LIN {X 0,Y 199.613,Z 910.43,A -85,B 0,C 180,E1 -21655.713,E2 -21655.713} C_VEL
LIN {X 0,Y 199.947,Z 910.384,A -85,B 0,C 180,E1 -21661.488,E2 -21661.488} C_VEL
LIN {X 0,Y 200.051,Z 910.436,A -85,B 0,C 180,E1 -21662.505,E2 -21662.505} C_VEL
LIN {X 0,Y 201.275,Z 916.976,A -85,B 0,C 180,E1 -21665.835,E2 -21665.835} C_VEL
LIN {X 0,Y 200.308,Z 922.874,A -85,B 0,C 180,E1 -21668.72,E2 -21668.72} C_VEL
LIN {X 0,Y 200.829,Z 941.062,A -85,B 0,C 180,E1 -21669.859,E2 -21669.859} C_VEL
LIN {X 0,Y 202.996,Z 965.944,A -85,B 0,C 180,E1 -21671.404,E2 -21671.404} C_VEL
LIN {X 0,Y 201.928,Z 1002.393,A -85,B 0,C 180,E1 -21673.768,E2 -21673.768} C_VEL
LIN {X 0,Y 201.253,Z 1013.208,A -85,B 0,C 180,E1 -21674.803,E2 -21674.803} C_VEL
LIN {X 0,Y 200.691,Z 1016.798,A -85,B 0,C 180,E1 -21675.235,E2 -21675.235} C_VEL
LIN {X 0,Y 198.329,Z 1023.524,A -85,B 0,C 180,E1 -21676.228,E2 -21676.228} C_VEL
LIN {X 0,Y 193.611,Z 1034.526,A -85,B 0,C 180,E1 -21678.361,E2 -21678.361} C_VEL
LIN {X 0,Y 192.718,Z 1039.161,A -85,B 0,C 180,E1 -21679.407,E2 -21679.407} C_VEL
LIN {X 0,Y 192.269,Z 1046.284,A -85,B 0,C 180,E1 -21681.169,E2 -21681.169} C_VEL
LIN {X 0,Y 191.944,Z 1053.424,A -85,B 0,C 180,E1 -21683.283,E2 -21683.283} C_VEL
LIN {X 0,Y 191.706,Z 1060.328,A -85,B 0,C 180,E1 -21685.795,E2 -21685.795} C_VEL
LIN {X 0,Y 191.489,Z 1064.888,A -85,B 0,C 180,E1 -21687.896,E2 -21687.896} C_VEL
LIN {X 0,Y 191.203,Z 1070.236,A -85,B 0,C 180,E1 -21691.053,E2 -21691.053} C_VEL
LIN {X 0,Y 190.853,Z 1074.06,A -85,B 0,C 180,E1 -21694.223,E2 -21694.223} C_VEL
LIN {X 0,Y 190.769,Z 1075.958,A -85,B 0,C 180,E1 -21696.345,E2 -21696.345} C_VEL
LIN {X 0,Y 191.01,Z 1077.321,A -85,B 0,C 180,E1 -21698.463,E2 -21698.463} C_VEL
LIN {X 0,Y 191.494,Z 1078.158,A -85,B 0,C 180,E1 -21700.574,E2 -21700.574} C_VEL
LIN {X 0,Y 192.366,Z 1078.612,A -85,B 0,C 180,E1 -21702.662,E2 -21702.662} C_VEL
LIN {X 0,Y 193.533,Z 1078.656,A -85,B 0,C 180,E1 -21704.726,E2 -21704.726} C_VEL
LIN {X 0,Y 195.065,Z 1078.141,A -85,B 0,C 180,E1 -21706.752,E2 -21706.752} C_VEL
LIN {X 0,Y 196.852,Z 1077.188,A -85,B 0,C 180,E1 -21708.742,E2 -21708.742} C_VEL
LIN {X 0,Y 198.954,Z 1075.838,A -85,B 0,C 180,E1 -21710.686,E2 -21710.686} C_VEL
LIN {X 0,Y 202.69,Z 1072.86,A -85,B 0,C 180,E1 -21713.5,E2 -21713.5} C_VEL
LIN {X 0,Y 207.145,Z 1068.693,A -85,B 0,C 180,E1 -21716.171,E2 -21716.171} C_VEL
LIN {X 0,Y 212.234,Z 1063.329,A -85,B 0,C 180,E1 -21718.696,E2 -21718.696} C_VEL
LIN {X 0,Y 217.894,Z 1056.459,A -85,B 0,C 180,E1 -21721.069,E2 -21721.069} C_VEL
LIN {X 0,Y 223.018,Z 1049.383,A -85,B 0,C 180,E1 -21722.929,E2 -21722.929} C_VEL
LIN {X 0,Y 227.532,Z 1042.512,A -85,B 0,C 180,E1 -21724.312,E2 -21724.312} C_VEL
LIN {X 0,Y 232.833,Z 1033.277,A -85,B 0,C 180,E1 -21725.791,E2 -21725.791} C_VEL
LIN {X 0,Y 237.843,Z 1023.421,A -85,B 0,C 180,E1 -21726.993,E2 -21726.993} C_VEL
LIN {X 0,Y 242.457,Z 1012.13,A -85,B 0,C 180,E1 -21728.039,E2 -21728.039} C_VEL
LIN {X 0,Y 246.47,Z 1000.194,A -85,B 0,C 180,E1 -21728.853,E2 -21728.853} C_VEL
LIN {X 0,Y 248.933,Z 990.741,A -85,B 0,C 180,E1 -21729.395,E2 -21729.395} C_VEL
LIN {X 0,Y 248.237,Z 987.091,A -85,B 0,C 180,E1 -21731.284,E2 -21731.284} C_VEL
LIN {X 0,Y 247.848,Z 983.63,A -85,B 0,C 180,E1 -21734.105,E2 -21734.105} C_VEL
LIN {X 0,Y 247.778,Z 983.164,A -85,B 0,C 180,E1 -21735.162,E2 -21735.162} C_VEL
LIN {X 0,Y 248.134,Z 983.137,A -85,B 0,C 180,E1 -21737.635,E2 -21737.635} C_VEL
LIN {X 0,Y 249.346,Z 985.54,A -85,B 0,C 180,E1 -21740.596,E2 -21740.596} C_VEL
LIN {X 0,Y 249.596,Z 986.288,A -85,B 0,C 180,E1 -21741.087,E2 -21741.087} C_VEL
LIN {X 0,Y 246.318,Z 998.437,A -85,B 0,C 180,E1 -21741.85,E2 -21741.85} C_VEL
LIN {X 0,Y 241.936,Z 1011.048,A -85,B 0,C 180,E1 -21742.932,E2 -21742.932} C_VEL
LIN {X 0,Y 237.247,Z 1021.654,A -85,B 0,C 180,E1 -21744.194,E2 -21744.194} C_VEL
LIN {X 0,Y 232.693,Z 1030.307,A -85,B 0,C 180,E1 -21745.508,E2 -21745.508} C_VEL
LIN {X 0,Y 226.976,Z 1039.66,A -85,B 0,C 180,E1 -21747.356,E2 -21747.356} C_VEL
LIN {X 0,Y 222.227,Z 1046.268,A -85,B 0,C 180,E1 -21749.076,E2 -21749.076} C_VEL
LIN {X 0,Y 217.511,Z 1052.076,A -85,B 0,C 180,E1 -21751.01,E2 -21751.01} C_VEL
LIN {X 0,Y 212.195,Z 1057.722,A -85,B 0,C 180,E1 -21753.442,E2 -21753.442} C_VEL
LIN {X 0,Y 207.462,Z 1061.91,A -85,B 0,C 180,E1 -21756.015,E2 -21756.015} C_VEL
LIN {X 0,Y 204.546,Z 1064.015,A -85,B 0,C 180,E1 -21757.794,E2 -21757.794} C_VEL
LIN {X 0,Y 201.845,Z 1065.571,A -85,B 0,C 180,E1 -21759.624,E2 -21759.624} C_VEL
LIN {X 0,Y 199.438,Z 1066.666,A -85,B 0,C 180,E1 -21761.51,E2 -21761.51} C_VEL
LIN {X 0,Y 197.357,Z 1067.342,A -85,B 0,C 180,E1 -21763.449,E2 -21763.449} C_VEL
LIN {X 0,Y 195.619,Z 1067.461,A -85,B 0,C 180,E1 -21765.435,E2 -21765.435} C_VEL
LIN {X 0,Y 194.191,Z 1067.076,A -85,B 0,C 180,E1 -21767.459,E2 -21767.459} C_VEL
LIN {X 0,Y 192.9,Z 1066.286,A -85,B 0,C 180,E1 -21769.505,E2 -21769.505} C_VEL
LIN {X 0,Y 191.826,Z 1065.04,A -85,B 0,C 180,E1 -21771.574,E2 -21771.574} C_VEL
LIN {X 0,Y 190.973,Z 1062.137,A -85,B 0,C 180,E1 -21774.722,E2 -21774.722} C_VEL
LIN {X 0,Y 190.674,Z 1058.072,A -85,B 0,C 180,E1 -21777.889,E2 -21777.889} C_VEL
LIN {X 0,Y 190.619,Z 1052.596,A -85,B 0,C 180,E1 -21781.057,E2 -21781.057} C_VEL
LIN {X 0,Y 190.791,Z 1046.812,A -85,B 0,C 180,E1 -21783.697,E2 -21783.697} C_VEL
LIN {X 0,Y 191.238,Z 1038.6,A -85,B 0,C 180,E1 -21786.649,E2 -21786.649} C_VEL
LIN {X 0,Y 191.776,Z 1030.551,A -85,B 0,C 180,E1 -21788.961,E2 -21788.961} C_VEL
LIN {X 0,Y 192.397,Z 1021.548,A -85,B 0,C 180,E1 -21791.057,E2 -21791.057} C_VEL
LIN {X 0,Y 193.113,Z 1011.82,A -85,B 0,C 180,E1 -21792.881,E2 -21792.881} C_VEL
LIN {X 0,Y 193.848,Z 1001.106,A -85,B 0,C 180,E1 -21794.434,E2 -21794.434} C_VEL
LIN {X 0,Y 194.455,Z 989.47,A -85,B 0,C 180,E1 -21795.729,E2 -21795.729} C_VEL
LIN {X 0,Y 195.048,Z 973.997,A -85,B 0,C 180,E1 -21796.89,E2 -21796.89} C_VEL
LIN {X 0,Y 196.308,Z 933.852,A -85,B 0,C 180,E1 -21799.526,E2 -21799.526} C_VEL
LIN {X 0,Y 193.913,Z 916.288,A -85,B 0,C 180,E1 -21800.666,E2 -21800.666} C_VEL
LIN {X 0,Y 192.915,Z 911.253,A -85,B 0,C 180,E1 -21801.025,E2 -21801.025} C_VEL
LIN {X 0,Y 192.57,Z 911.308,A -85,B 0,C 180,E1 -21805.974,E2 -21805.974} C_VEL
LIN {X 0,Y 192.602,Z 911.303,A -85,B 0,C 180,E1 -21808.866,E2 -21808.866} C_VEL
LIN {X 0,Y 192.596,Z 911.306,A -85,B 0,C 180,E1 -21813.188,E2 -21813.188} C_VEL
LIN {X 0,Y 192.542,Z 911.308,A -85,B 0,C 180,E1 -21818.355,E2 -21818.355} C_VEL
LIN {X 0,Y 192.486,Z 911.319,A -85,B 0,C 180,E1 -21823.094,E2 -21823.094} C_VEL
LIN {X 0,Y 192.488,Z 911.316,A -85,B 0,C 180,E1 -21826.907,E2 -21826.907} C_VEL
LIN {X 0,Y 192.544,Z 911.311,A -85,B 0,C 180,E1 -21831.647,E2 -21831.647} C_VEL
LIN {X 0,Y 192.598,Z 911.301,A -85,B 0,C 180,E1 -21836.814,E2 -21836.814} C_VEL
LIN {X 0,Y 192.624,Z 911.301,A -85,B 0,C 180,E1 -21841.686,E2 -21841.686} C_VEL
LIN {X 0,Y 192.674,Z 911.292,A -85,B 0,C 180,E1 -21846.345,E2 -21846.345} C_VEL
LIN {X 0,Y 192.698,Z 911.294,A -85,B 0,C 180,E1 -21851.492,E2 -21851.492} C_VEL
LIN {X 0,Y 192.74,Z 911.286,A -85,B 0,C 180,E1 -21855.212,E2 -21855.212} C_VEL
LIN {X 0,Y 192.95,Z 911.264,A -85,B 0,C 180,E1 -21859.567,E2 -21859.567} C_VEL
LIN {X 0,Y 192.967,Z 911.258,A -85,B 0,C 180,E1 -21863.728,E2 -21863.728} C_VEL
LIN {X 0,Y 193.212,Z 911.23,A -85,B 0,C 180,E1 -21867.916,E2 -21867.916} C_VEL
LIN {X 0,Y 193.414,Z 911.207,A -85,B 0,C 180,E1 -21870,E2 -21870} C_VEL
LIN {X 0,Y 192.921,Z 911.263,A -85,B 0,C 180,E1 -21874.179,E2 -21874.179} C_VEL
LIN {X 0,Y 193.03,Z 911.254,A -85,B 0,C 180,E1 -21878.374,E2 -21878.374} C_VEL
LIN {X 0,Y 192.781,Z 911.28,A -85,B 0,C 180,E1 -21882.635,E2 -21882.635} C_VEL
LIN {X 0,Y 192.699,Z 911.294,A -85,B 0,C 180,E1 -21888.508,E2 -21888.508} C_VEL
LIN {X 0,Y 192.615,Z 911.299,A -85,B 0,C 180,E1 -21894.189,E2 -21894.189} C_VEL
LIN {X 0,Y 192.605,Z 911.305,A -85,B 0,C 180,E1 -21898.865,E2 -21898.865} C_VEL
LIN {X 0,Y 192.599,Z 911.301,A -85,B 0,C 180,E1 -21903.186,E2 -21903.186} C_VEL
LIN {X 0,Y 192.546,Z 911.311,A -85,B 0,C 180,E1 -21908.354,E2 -21908.354} C_VEL
LIN {X 0,Y 192.49,Z 911.315,A -85,B 0,C 180,E1 -21913.093,E2 -21913.093} C_VEL
LIN {X 0,Y 192.49,Z 911.318,A -85,B 0,C 180,E1 -21916.906,E2 -21916.906} C_VEL
LIN {X 0,Y 192.546,Z 911.307,A -85,B 0,C 180,E1 -21921.645,E2 -21921.645} C_VEL
LIN {X 0,Y 192.598,Z 911.305,A -85,B 0,C 180,E1 -21926.813,E2 -21926.813} C_VEL
LIN {X 0,Y 192.623,Z 911.299,A -85,B 0,C 180,E1 -21931.684,E2 -21931.684} C_VEL
LIN {X 0,Y 192.66,Z 911.297,A -85,B 0,C 180,E1 -21936.341,E2 -21936.341} C_VEL
LIN {X 0,Y 192.698,Z 911.293,A -85,B 0,C 180,E1 -21941.491,E2 -21941.491} C_VEL
LIN {X 0,Y 192.721,Z 911.292,A -85,B 0,C 180,E1 -21945.209,E2 -21945.209} C_VEL
LIN {X 0,Y 192.949,Z 911.26,A -85,B 0,C 180,E1 -21949.566,E2 -21949.566} C_VEL
LIN {X 0,Y 192.965,Z 911.262,A -85,B 0,C 180,E1 -21953.726,E2 -21953.726} C_VEL
LIN {X 0,Y 193.21,Z 911.226,A -85,B 0,C 180,E1 -21957.914,E2 -21957.914} C_VEL
LIN {X 0,Y 193.412,Z 911.204,A -85,B 0,C 180,E1 -21959.999,E2 -21959.999} C_VEL
LIN {X 0,Y 192.918,Z 911.267,A -85,B 0,C 180,E1 -21964.177,E2 -21964.177} C_VEL
LIN {X 0,Y 193.023,Z 911.251,A -85,B 0,C 180,E1 -21968.373,E2 -21968.373} C_VEL
LIN {X 0,Y 192.782,Z 911.284,A -85,B 0,C 180,E1 -21972.634,E2 -21972.634} C_VEL
LIN {X 0,Y 192.704,Z 911.291,A -85,B 0,C 180,E1 -21976.963,E2 -21976.963} C_VEL
LIN {X 0,Y 192.573,Z 911.309,A -85,B 0,C 180,E1 -21981.404,E2 -21981.404} C_VEL
LIN {X 0,Y 192.611,Z 911.3,A -85,B 0,C 180,E1 -21984.188,E2 -21984.188} C_VEL
LIN {X 0,Y 192.601,Z 911.305,A -85,B 0,C 180,E1 -21988.864,E2 -21988.864} C_VEL
LIN {X 0,Y 192.595,Z 911.306,A -85,B 0,C 180,E1 -21993.186,E2 -21993.186} C_VEL
LIN {X 0,Y 192.541,Z 911.312,A -85,B 0,C 180,E1 -21998.353,E2 -21998.353} C_VEL
LIN {X 0,Y 192.485,Z 911.315,A -85,B 0,C 180,E1 -22003.093,E2 -22003.093} C_VEL
LIN {X 0,Y 192.485,Z 911.318,A -85,B 0,C 180,E1 -22006.905,E2 -22006.905} C_VEL
LIN {X 0,Y 192.541,Z 911.31,A -85,B 0,C 180,E1 -22011.645,E2 -22011.645} C_VEL
LIN {X 0,Y 192.599,Z 911.307,A -85,B 0,C 180,E1 -22016.814,E2 -22016.814} C_VEL
LIN {X 0,Y 193.061,Z 911.351,A -85,B 0,C 180,E1 -22022.786,E2 -22022.786} C_VEL
LIN {X 0,Y 194.169,Z 916.994,A -85,B 0,C 180,E1 -22025.773,E2 -22025.773} C_VEL
LIN {X 0,Y 193.24,Z 922.433,A -85,B 0,C 180,E1 -22028.602,E2 -22028.602} C_VEL
LIN {X 0,Y 193.68,Z 940.397,A -85,B 0,C 180,E1 -22029.776,E2 -22029.776} C_VEL
LIN {X 0,Y 195.896,Z 965.867,A -85,B 0,C 180,E1 -22031.433,E2 -22031.433} C_VEL
LIN {X 0,Y 194.873,Z 1001.979,A -85,B 0,C 180,E1 -22033.904,E2 -22033.904} C_VEL
LIN {X 0,Y 194.128,Z 1014.314,A -85,B 0,C 180,E1 -22035.185,E2 -22035.185} C_VEL
LIN {X 0,Y 193.646,Z 1024.555,A -85,B 0,C 180,E1 -22036.622,E2 -22036.622} C_VEL
LIN {X 0,Y 192.992,Z 1034.779,A -85,B 0,C 180,E1 -22038.446,E2 -22038.446} C_VEL
LIN {X 0,Y 192.718,Z 1039.161,A -85,B 0,C 180,E1 -22039.407,E2 -22039.407} C_VEL
LIN {X 0,Y 191.84,Z 1043.702,A -85,B 0,C 180,E1 -22040.518,E2 -22040.518} C_VEL
LIN {X 0,Y 190.093,Z 1047.709,A -85,B 0,C 180,E1 -22041.719,E2 -22041.719} C_VEL
LIN {X 0,Y 185.624,Z 1056.056,A -85,B 0,C 180,E1 -22044.869,E2 -22044.869} C_VEL
LIN {X 0,Y 184.797,Z 1059.5,A -85,B 0,C 180,E1 -22046.348,E2 -22046.348} C_VEL
LIN {X 0,Y 184.526,Z 1064.875,A -85,B 0,C 180,E1 -22048.908,E2 -22048.908} C_VEL
LIN {X 0,Y 184.314,Z 1068.52,A -85,B 0,C 180,E1 -22051.092,E2 -22051.092} C_VEL
LIN {X 0,Y 183.898,Z 1072.684,A -85,B 0,C 180,E1 -22054.383,E2 -22054.383} C_VEL
LIN {X 0,Y 183.818,Z 1074.699,A -85,B 0,C 180,E1 -22056.586,E2 -22056.586} C_VEL
LIN {X 0,Y 184.05,Z 1076.245,A -85,B 0,C 180,E1 -22058.785,E2 -22058.785} C_VEL
LIN {X 0,Y 184.551,Z 1077.372,A -85,B 0,C 180,E1 -22060.976,E2 -22060.976} C_VEL
LIN {X 0,Y 185.461,Z 1078.068,A -85,B 0,C 180,E1 -22063.142,E2 -22063.142} C_VEL
LIN {X 0,Y 186.677,Z 1078.217,A -85,B 0,C 180,E1 -22065.28,E2 -22065.28} C_VEL
LIN {X 0,Y 190.141,Z 1077.365,A -85,B 0,C 180,E1 -22069.43,E2 -22069.43} C_VEL
LIN {X 0,Y 192.337,Z 1076.209,A -85,B 0,C 180,E1 -22071.432,E2 -22071.432} C_VEL
LIN {X 0,Y 196.255,Z 1073.673,A -85,B 0,C 180,E1 -22074.319,E2 -22074.319} C_VEL
LIN {X 0,Y 200.896,Z 1070.053,A -85,B 0,C 180,E1 -22077.051,E2 -22077.051} C_VEL
LIN {X 0,Y 206.16,Z 1065.117,A -85,B 0,C 180,E1 -22079.624,E2 -22079.624} C_VEL
LIN {X 0,Y 210.987,Z 1060.06,A -85,B 0,C 180,E1 -22081.643,E2 -22081.643} C_VEL
LIN {X 0,Y 216.211,Z 1053.859,A -85,B 0,C 180,E1 -22083.545,E2 -22083.545} C_VEL
LIN {X 0,Y 221.935,Z 1046.324,A -85,B 0,C 180,E1 -22085.304,E2 -22085.304} C_VEL
LIN {X 0,Y 228.294,Z 1036.758,A -85,B 0,C 180,E1 -22087.002,E2 -22087.002} C_VEL
LIN {X 0,Y 233.954,Z 1026.535,A -85,B 0,C 180,E1 -22088.323,E2 -22088.323} C_VEL
LIN {X 0,Y 239.092,Z 1015.776,A -85,B 0,C 180,E1 -22089.395,E2 -22089.395} C_VEL
LIN {X 0,Y 243.435,Z 1004.387,A -85,B 0,C 180,E1 -22090.233,E2 -22090.233} C_VEL
LIN {X 0,Y 246.188,Z 995.227,A -85,B 0,C 180,E1 -22090.794,E2 -22090.794} C_VEL
LIN {X 0,Y 246.017,Z 993.347,A -85,B 0,C 180,E1 -22091.921,E2 -22091.921} C_VEL
LIN {X 0,Y 245.926,Z 990.354,A -85,B 0,C 180,E1 -22094.403,E2 -22094.403} C_VEL
LIN {X 0,Y 246.067,Z 989.856,A -85,B 0,C 180,E1 -22096.728,E2 -22096.728} C_VEL
LIN {X 0,Y 246.307,Z 990.295,A -85,B 0,C 180,E1 -22098.048,E2 -22098.048} C_VEL
LIN {X 0,Y 246.851,Z 991.576,A -85,B 0,C 180,E1 -22099.769,E2 -22099.769} C_VEL
LIN {X 0,Y 242.902,Z 1004.222,A -85,B 0,C 180,E1 -22100.622,E2 -22100.622} C_VEL
LIN {X 0,Y 238.748,Z 1014.42,A -85,B 0,C 180,E1 -22101.588,E2 -22101.588} C_VEL
LIN {X 0,Y 233.909,Z 1024.259,A -85,B 0,C 180,E1 -22102.796,E2 -22102.796} C_VEL
LIN {X 0,Y 228.57,Z 1033.478,A -85,B 0,C 180,E1 -22104.254,E2 -22104.254} C_VEL
LIN {X 0,Y 224.029,Z 1040.184,A -85,B 0,C 180,E1 -22105.621,E2 -22105.621} C_VEL
LIN {X 0,Y 218.648,Z 1047.117,A -85,B 0,C 180,E1 -22107.426,E2 -22107.426} C_VEL
LIN {X 0,Y 213.847,Z 1052.566,A -85,B 0,C 180,E1 -22109.218,E2 -22109.218} C_VEL
LIN {X 0,Y 207.879,Z 1058.36,A -85,B 0,C 180,E1 -22111.751,E2 -22111.751} C_VEL
LIN {X 0,Y 202.523,Z 1062.642,A -85,B 0,C 180,E1 -22114.456,E2 -22114.456} C_VEL
LIN {X 0,Y 198.095,Z 1065.348,A -85,B 0,C 180,E1 -22117.03,E2 -22117.03} C_VEL
LIN {X 0,Y 195.309,Z 1066.722,A -85,B 0,C 180,E1 -22118.911,E2 -22118.911} C_VEL
LIN {X 0,Y 192.768,Z 1067.514,A -85,B 0,C 180,E1 -22120.846,E2 -22120.846} C_VEL
LIN {X 0,Y 190.602,Z 1067.84,A -85,B 0,C 180,E1 -22122.845,E2 -22122.845} C_VEL
LIN {X 0,Y 188.778,Z 1067.767,A -85,B 0,C 180,E1 -22124.895,E2 -22124.895} C_VEL
LIN {X 0,Y 187.286,Z 1067.222,A -85,B 0,C 180,E1 -22126.989,E2 -22126.989} C_VEL
LIN {X 0,Y 185.935,Z 1066.121,A -85,B 0,C 180,E1 -22129.107,E2 -22129.107} C_VEL
LIN {X 0,Y 184.643,Z 1064.185,A -85,B 0,C 180,E1 -22131.74,E2 -22131.74} C_VEL
LIN {X 0,Y 183.951,Z 1061.382,A -85,B 0,C 180,E1 -22134.52,E2 -22134.52} C_VEL
LIN {X 0,Y 183.674,Z 1056.99,A -85,B 0,C 180,E1 -22137.808,E2 -22137.808} C_VEL
LIN {X 0,Y 183.649,Z 1051.201,A -85,B 0,C 180,E1 -22141.097,E2 -22141.097} C_VEL
LIN {X 0,Y 183.837,Z 1044.932,A -85,B 0,C 180,E1 -22143.837,E2 -22143.837} C_VEL
LIN {X 0,Y 184.283,Z 1037.182,A -85,B 0,C 180,E1 -22146.571,E2 -22146.571} C_VEL
LIN {X 0,Y 184.847,Z 1028.643,A -85,B 0,C 180,E1 -22149.024,E2 -22149.024} C_VEL
LIN {X 0,Y 185.591,Z 1017.821,A -85,B 0,C 180,E1 -22151.468,E2 -22151.468} C_VEL
LIN {X 0,Y 186.206,Z 1008.819,A -85,B 0,C 180,E1 -22153.09,E2 -22153.09} C_VEL
LIN {X 0,Y 186.966,Z 997.471,A -85,B 0,C 180,E1 -22154.699,E2 -22154.699} C_VEL
LIN {X 0,Y 187.473,Z 985.392,A -85,B 0,C 180,E1 -22155.911,E2 -22155.911} C_VEL
LIN {X 0,Y 188.831,Z 947.508,A -85,B 0,C 180,E1 -22158.584,E2 -22158.584} C_VEL
LIN {X 0,Y 189.199,Z 934.016,A -85,B 0,C 180,E1 -22159.506,E2 -22159.506} C_VEL
LIN {X 0,Y 186.804,Z 916.793,A -85,B 0,C 180,E1 -22160.665,E2 -22160.665} C_VEL
LIN {X 0,Y 185.884,Z 912.129,A -85,B 0,C 180,E1 -22161.027,E2 -22161.027} C_VEL
LIN {X 0,Y 185.509,Z 912.19,A -85,B 0,C 180,E1 -22167.042,E2 -22167.042} C_VEL
LIN {X 0,Y 185.545,Z 912.18,A -85,B 0,C 180,E1 -22169.5,E2 -22169.5} C_VEL
LIN {X 0,Y 185.498,Z 912.189,A -85,B 0,C 180,E1 -22174.634,E2 -22174.634} C_VEL
LIN {X 0,Y 185.501,Z 912.189,A -85,B 0,C 180,E1 -22177.316,E2 -22177.316} C_VEL
LIN {X 0,Y 185.462,Z 912.191,A -85,B 0,C 180,E1 -22180.722,E2 -22180.722} C_VEL
LIN {X 0,Y 185.458,Z 912.195,A -85,B 0,C 180,E1 -22186.057,E2 -22186.057} C_VEL
LIN {X 0,Y 185.459,Z 912.192,A -85,B 0,C 180,E1 -22189.893,E2 -22189.893} C_VEL
LIN {X 0,Y 185.503,Z 912.19,A -85,B 0,C 180,E1 -22192.715,E2 -22192.715} C_VEL
LIN {X 0,Y 185.534,Z 912.18,A -85,B 0,C 180,E1 -22197.973,E2 -22197.973} C_VEL
LIN {X 0,Y 185.55,Z 912.184,A -85,B 0,C 180,E1 -22200.596,E2 -22200.596} C_VEL
LIN {X 0,Y 185.584,Z 912.176,A -85,B 0,C 180,E1 -22205.382,E2 -22205.382} C_VEL
LIN {X 0,Y 185.629,Z 912.176,A -85,B 0,C 180,E1 -22211.179,E2 -22211.179} C_VEL
LIN {X 0,Y 185.669,Z 912.166,A -85,B 0,C 180,E1 -22214.635,E2 -22214.635} C_VEL
LIN {X 0,Y 185.893,Z 912.142,A -85,B 0,C 180,E1 -22219.419,E2 -22219.419} C_VEL
LIN {X 0,Y 185.933,Z 912.136,A -85,B 0,C 180,E1 -22223.489,E2 -22223.489} C_VEL
LIN {X 0,Y 186.379,Z 912.083,A -85,B 0,C 180,E1 -22230,E2 -22230} C_VEL
LIN {X 0,Y 185.932,Z 912.136,A -85,B 0,C 180,E1 -22236.512,E2 -22236.512} C_VEL
LIN {X 0,Y 185.893,Z 912.142,A -85,B 0,C 180,E1 -22240.581,E2 -22240.581} C_VEL
LIN {X 0,Y 185.646,Z 912.169,A -85,B 0,C 180,E1 -22245.367,E2 -22245.367} C_VEL
LIN {X 0,Y 185.629,Z 912.176,A -85,B 0,C 180,E1 -22248.821,E2 -22248.821} C_VEL
LIN {X 0,Y 185.549,Z 912.18,A -85,B 0,C 180,E1 -22254.624,E2 -22254.624} C_VEL
LIN {X 0,Y 185.548,Z 912.184,A -85,B 0,C 180,E1 -22259.499,E2 -22259.499} C_VEL
LIN {X 0,Y 185.501,Z 912.187,A -85,B 0,C 180,E1 -22264.632,E2 -22264.632} C_VEL
LIN {X 0,Y 185.504,Z 912.19,A -85,B 0,C 180,E1 -22267.314,E2 -22267.314} C_VEL
LIN {X 0,Y 185.466,Z 912.189,A -85,B 0,C 180,E1 -22270.721,E2 -22270.721} C_VEL
LIN {X 0,Y 185.46,Z 912.197,A -85,B 0,C 180,E1 -22276.055,E2 -22276.055} C_VEL
LIN {X 0,Y 185.461,Z 912.193,A -85,B 0,C 180,E1 -22279.892,E2 -22279.892} C_VEL
LIN {X 0,Y 185.504,Z 912.189,A -85,B 0,C 180,E1 -22282.713,E2 -22282.713} C_VEL
LIN {X 0,Y 185.534,Z 912.184,A -85,B 0,C 180,E1 -22287.972,E2 -22287.972} C_VEL
LIN {X 0,Y 185.55,Z 912.18,A -85,B 0,C 180,E1 -22290.595,E2 -22290.595} C_VEL
LIN {X 0,Y 185.548,Z 912.184,A -85,B 0,C 180,E1 -22295.376,E2 -22295.376} C_VEL
LIN {X 0,Y 185.628,Z 912.173,A -85,B 0,C 180,E1 -22301.178,E2 -22301.178} C_VEL
LIN {X 0,Y 185.707,Z 912.162,A -85,B 0,C 180,E1 -22306.874,E2 -22306.874} C_VEL
LIN {X 0,Y 185.978,Z 912.13,A -85,B 0,C 180,E1 -22311.305,E2 -22311.305} C_VEL
LIN {X 0,Y 186.158,Z 912.104,A -85,B 0,C 180,E1 -22317.835,E2 -22317.835} C_VEL
LIN {X 0,Y 186.377,Z 912.08,A -85,B 0,C 180,E1 -22319.999,E2 -22319.999} C_VEL
LIN {X 0,Y 185.927,Z 912.133,A -85,B 0,C 180,E1 -22326.51,E2 -22326.51} C_VEL
LIN {X 0,Y 185.89,Z 912.143,A -85,B 0,C 180,E1 -22330.58,E2 -22330.58} C_VEL
LIN {X 0,Y 185.652,Z 912.166,A -85,B 0,C 180,E1 -22335.365,E2 -22335.365} C_VEL
LIN {X 0,Y 185.626,Z 912.174,A -85,B 0,C 180,E1 -22338.82,E2 -22338.82} C_VEL
LIN {X 0,Y 185.545,Z 912.181,A -85,B 0,C 180,E1 -22344.622,E2 -22344.622} C_VEL
LIN {X 0,Y 185.544,Z 912.186,A -85,B 0,C 180,E1 -22349.498,E2 -22349.498} C_VEL
LIN {X 0,Y 185.497,Z 912.184,A -85,B 0,C 180,E1 -22354.631,E2 -22354.631} C_VEL
LIN {X 0,Y 185.499,Z 912.189,A -85,B 0,C 180,E1 -22357.314,E2 -22357.314} C_VEL
LIN {X 0,Y 185.462,Z 912.193,A -85,B 0,C 180,E1 -22360.72,E2 -22360.72} C_VEL
LIN {X 0,Y 185.456,Z 912.195,A -85,B 0,C 180,E1 -22366.055,E2 -22366.055} C_VEL
LIN {X 0,Y 185.456,Z 912.196,A -85,B 0,C 180,E1 -22369.891,E2 -22369.891} C_VEL
LIN {X 0,Y 185.499,Z 912.185,A -85,B 0,C 180,E1 -22372.713,E2 -22372.713} C_VEL
LIN {X 0,Y 185.575,Z 912.18,A -85,B 0,C 180,E1 -22377.98,E2 -22377.98} C_VEL
LIN {X 0,Y 186.041,Z 912.134,A -85,B 0,C 180,E1 -22383.043,E2 -22383.043} C_VEL
LIN {X 0,Y 186.989,Z 916.741,A -85,B 0,C 180,E1 -22385.579,E2 -22385.579} C_VEL
LIN {X 0,Y 186.152,Z 922.334,A -85,B 0,C 180,E1 -22388.547,E2 -22388.547} C_VEL
LIN {X 0,Y 186.629,Z 941.521,A -85,B 0,C 180,E1 -22389.867,E2 -22389.867} C_VEL
LIN {X 0,Y 188.81,Z 966.35,A -85,B 0,C 180,E1 -22391.555,E2 -22391.555} C_VEL
LIN {X 0,Y 187.807,Z 1001.86,A -85,B 0,C 180,E1 -22394.118,E2 -22394.118} C_VEL
LIN {X 0,Y 187.082,Z 1014.101,A -85,B 0,C 180,E1 -22395.45,E2 -22395.45} C_VEL
LIN {X 0,Y 186.609,Z 1024.295,A -85,B 0,C 180,E1 -22396.94,E2 -22396.94} C_VEL
LIN {X 0,Y 185.971,Z 1034.491,A -85,B 0,C 180,E1 -22398.832,E2 -22398.832} C_VEL
LIN {X 0,Y 185.473,Z 1042.984,A -85,B 0,C 180,E1 -22400.843,E2 -22400.843} C_VEL
LIN {X 0,Y 185.117,Z 1050.175,A -85,B 0,C 180,E1 -22402.935,E2 -22402.935} C_VEL
LIN {X 0,Y 184.915,Z 1056.366,A -85,B 0,C 180,E1 -22405.094,E2 -22405.094} C_VEL
LIN {X 0,Y 184.797,Z 1059.5,A -85,B 0,C 180,E1 -22406.348,E2 -22406.348} C_VEL
LIN {X 0,Y 183.946,Z 1062.661,A -85,B 0,C 180,E1 -22407.871,E2 -22407.871} C_VEL
LIN {X 0,Y 182.207,Z 1065.218,A -85,B 0,C 180,E1 -22409.462,E2 -22409.462} C_VEL
LIN {X 0,Y 178.237,Z 1069.314,A -85,B 0,C 180,E1 -22412.853,E2 -22412.853} C_VEL
LIN {X 0,Y 177.065,Z 1071.181,A -85,B 0,C 180,E1 -22414.66,E2 -22414.66} C_VEL
LIN {X 0,Y 176.93,Z 1071.85,A -85,B 0,C 180,E1 -22415.27,E2 -22415.27} C_VEL
LIN {X 0,Y 177.131,Z 1075.134,A -85,B 0,C 180,E1 -22419.131,E2 -22419.131} C_VEL
LIN {X 0,Y 177.645,Z 1076.441,A -85,B 0,C 180,E1 -22421.409,E2 -22421.409} C_VEL
LIN {X 0,Y 179.844,Z 1077.726,A -85,B 0,C 180,E1 -22425.875,E2 -22425.875} C_VEL
LIN {X 0,Y 181.515,Z 1077.786,A -85,B 0,C 180,E1 -22428.044,E2 -22428.044} C_VEL
LIN {X 0,Y 185.748,Z 1076.415,A -85,B 0,C 180,E1 -22432.232,E2 -22432.232} C_VEL
LIN {X 0,Y 188.366,Z 1075.181,A -85,B 0,C 180,E1 -22434.231,E2 -22434.231} C_VEL
LIN {X 0,Y 193.011,Z 1072.32,A -85,B 0,C 180,E1 -22437.075,E2 -22437.075} C_VEL
LIN {X 0,Y 198.268,Z 1068.366,A -85,B 0,C 180,E1 -22439.752,E2 -22439.752} C_VEL
LIN {X 0,Y 204.114,Z 1063.197,A -85,B 0,C 180,E1 -22442.255,E2 -22442.255} C_VEL
LIN {X 0,Y 211.688,Z 1055.492,A -85,B 0,C 180,E1 -22444.938,E2 -22444.938} C_VEL
LIN {X 0,Y 217.638,Z 1048.375,A -85,B 0,C 180,E1 -22446.684,E2 -22446.684} C_VEL
LIN {X 0,Y 224.464,Z 1039.022,A -85,B 0,C 180,E1 -22448.428,E2 -22448.428} C_VEL
LIN {X 0,Y 230.685,Z 1029.152,A -85,B 0,C 180,E1 -22449.775,E2 -22449.775} C_VEL
LIN {X 0,Y 236.796,Z 1017.209,A -85,B 0,C 180,E1 -22450.974,E2 -22450.974} C_VEL
LIN {X 0,Y 241.585,Z 1006.027,A -85,B 0,C 180,E1 -22451.811,E2 -22451.811} C_VEL
LIN {X 0,Y 243.512,Z 1000.473,A -85,B 0,C 180,E1 -22452.13,E2 -22452.13} C_VEL
LIN {X 0,Y 243.617,Z 999.565,A -85,B 0,C 180,E1 -22452.534,E2 -22452.534} C_VEL
LIN {X 0,Y 243.682,Z 997.94,A -85,B 0,C 180,E1 -22453.862,E2 -22453.862} C_VEL
LIN {X 0,Y 243.888,Z 996.666,A -85,B 0,C 180,E1 -22456.244,E2 -22456.244} C_VEL
LIN {X 0,Y 244.204,Z 997.405,A -85,B 0,C 180,E1 -22458.44,E2 -22458.44} C_VEL
LIN {X 0,Y 240.203,Z 1008.138,A -85,B 0,C 180,E1 -22459.233,E2 -22459.233} C_VEL
LIN {X 0,Y 235.252,Z 1018.903,A -85,B 0,C 180,E1 -22460.316,E2 -22460.316} C_VEL
LIN {X 0,Y 229.487,Z 1029.124,A -85,B 0,C 180,E1 -22461.674,E2 -22461.674} C_VEL
LIN {X 0,Y 224.556,Z 1036.55,A -85,B 0,C 180,E1 -22462.954,E2 -22462.954} C_VEL
LIN {X 0,Y 217.528,Z 1045.679,A -85,B 0,C 180,E1 -22465.008,E2 -22465.008} C_VEL
LIN {X 0,Y 211.983,Z 1051.678,A -85,B 0,C 180,E1 -22466.837,E2 -22466.837} C_VEL
LIN {X 0,Y 205.792,Z 1057.434,A -85,B 0,C 180,E1 -22469.186,E2 -22469.186} C_VEL
LIN {X 0,Y 200.896,Z 1061.269,A -85,B 0,C 180,E1 -22471.28,E2 -22471.28} C_VEL
LIN {X 0,Y 194.89,Z 1065.127,A -85,B 0,C 180,E1 -22474.36,E2 -22474.36} C_VEL
LIN {X 0,Y 191.695,Z 1066.597,A -85,B 0,C 180,E1 -22476.217,E2 -22476.217} C_VEL
LIN {X 0,Y 188.77,Z 1067.618,A -85,B 0,C 180,E1 -22478.143,E2 -22478.143} C_VEL
LIN {X 0,Y 186.131,Z 1068.231,A -85,B 0,C 180,E1 -22480.135,E2 -22480.135} C_VEL
LIN {X 0,Y 183.855,Z 1068.337,A -85,B 0,C 180,E1 -22482.194,E2 -22482.194} C_VEL
LIN {X 0,Y 180.383,Z 1067.112,A -85,B 0,C 180,E1 -22486.482,E2 -22486.482} C_VEL
LIN {X 0,Y 178.987,Z 1065.887,A -85,B 0,C 180,E1 -22488.679,E2 -22488.679} C_VEL
LIN {X 0,Y 177.524,Z 1063.295,A -85,B 0,C 180,E1 -22491.778,E2 -22491.778} C_VEL
LIN {X 0,Y 176.794,Z 1059.06,A -85,B 0,C 180,E1 -22495.441,E2 -22495.441} C_VEL
LIN {X 0,Y 176.625,Z 1053.778,A -85,B 0,C 180,E1 -22498.861,E2 -22498.861} C_VEL
LIN {X 0,Y 176.785,Z 1047.015,A -85,B 0,C 180,E1 -22502.279,E2 -22502.279} C_VEL
LIN {X 0,Y 177.117,Z 1038.771,A -85,B 0,C 180,E1 -22505.467,E2 -22505.467} C_VEL
LIN {X 0,Y 177.6,Z 1031.527,A -85,B 0,C 180,E1 -22507.735,E2 -22507.735} C_VEL
LIN {X 0,Y 178.262,Z 1021.803,A -85,B 0,C 180,E1 -22510.22,E2 -22510.22} C_VEL
LIN {X 0,Y 179.067,Z 1010.463,A -85,B 0,C 180,E1 -22512.467,E2 -22512.467} C_VEL
LIN {X 0,Y 179.799,Z 999.569,A -85,B 0,C 180,E1 -22514.142,E2 -22514.142} C_VEL
LIN {X 0,Y 180.396,Z 986.471,A -85,B 0,C 180,E1 -22515.609,E2 -22515.609} C_VEL
LIN {X 0,Y 181.67,Z 949.522,A -85,B 0,C 180,E1 -22518.394,E2 -22518.394} C_VEL
LIN {X 0,Y 182.084,Z 934.335,A -85,B 0,C 180,E1 -22519.473,E2 -22519.473} C_VEL
LIN {X 0,Y 179.789,Z 917.903,A -85,B 0,C 180,E1 -22520.633,E2 -22520.633} C_VEL
LIN {X 0,Y 178.835,Z 913.007,A -85,B 0,C 180,E1 -22521.015,E2 -22521.015} C_VEL
LIN {X 0,Y 178.487,Z 913.063,A -85,B 0,C 180,E1 -22525.668,E2 -22525.668} C_VEL
LIN {X 0,Y 178.461,Z 913.061,A -85,B 0,C 180,E1 -22530.795,E2 -22530.795} C_VEL
LIN {X 0,Y 178.484,Z 913.063,A -85,B 0,C 180,E1 -22534.219,E2 -22534.219} C_VEL
LIN {X 0,Y 178.388,Z 913.07,A -85,B 0,C 180,E1 -22539.078,E2 -22539.078} C_VEL
LIN {X 0,Y 178.395,Z 913.076,A -85,B 0,C 180,E1 -22542.048,E2 -22542.048} C_VEL
LIN {X 0,Y 178.393,Z 913.074,A -85,B 0,C 180,E1 -22545.166,E2 -22545.166} C_VEL
LIN {X 0,Y 178.4,Z 913.07,A -85,B 0,C 180,E1 -22548.462,E2 -22548.462} C_VEL
LIN {X 0,Y 178.421,Z 913.071,A -85,B 0,C 180,E1 -22553.783,E2 -22553.783} C_VEL
LIN {X 0,Y 178.487,Z 913.06,A -85,B 0,C 180,E1 -22556.547,E2 -22556.547} C_VEL
LIN {X 0,Y 178.447,Z 913.068,A -85,B 0,C 180,E1 -22561.796,E2 -22561.796} C_VEL
LIN {X 0,Y 178.519,Z 913.058,A -85,B 0,C 180,E1 -22564.89,E2 -22564.89} C_VEL
LIN {X 0,Y 178.612,Z 913.048,A -85,B 0,C 180,E1 -22571.653,E2 -22571.653} C_VEL
LIN {X 0,Y 178.646,Z 913.037,A -85,B 0,C 180,E1 -22576.347,E2 -22576.347} C_VEL
LIN {X 0,Y 178.91,Z 913.01,A -85,B 0,C 180,E1 -22580.96,E2 -22580.96} C_VEL
LIN {X 0,Y 178.821,Z 913.018,A -85,B 0,C 180,E1 -22585.492,E2 -22585.492} C_VEL
LIN {X 0,Y 179.344,Z 912.959,A -85,B 0,C 180,E1 -22590,E2 -22590} C_VEL
LIN {X 0,Y 178.898,Z 913.011,A -85,B 0,C 180,E1 -22596.769,E2 -22596.769} C_VEL
LIN {X 0,Y 178.838,Z 913.019,A -85,B 0,C 180,E1 -22600.742,E2 -22600.742} C_VEL
LIN {X 0,Y 178.574,Z 913.05,A -85,B 0,C 180,E1 -22605.992,E2 -22605.992} C_VEL
LIN {X 0,Y 178.559,Z 913.055,A -85,B 0,C 180,E1 -22609.152,E2 -22609.152} C_VEL
LIN {X 0,Y 178.47,Z 913.064,A -85,B 0,C 180,E1 -22615.076,E2 -22615.076} C_VEL
LIN {X 0,Y 178.464,Z 913.064,A -85,B 0,C 180,E1 -22620.794,E2 -22620.794} C_VEL
LIN {X 0,Y 178.487,Z 913.061,A -85,B 0,C 180,E1 -22624.218,E2 -22624.218} C_VEL
LIN {X 0,Y 178.391,Z 913.074,A -85,B 0,C 180,E1 -22629.076,E2 -22629.076} C_VEL
LIN {X 0,Y 178.398,Z 913.071,A -85,B 0,C 180,E1 -22632.046,E2 -22632.046} C_VEL
LIN {X 0,Y 178.396,Z 913.074,A -85,B 0,C 180,E1 -22635.164,E2 -22635.164} C_VEL
LIN {X 0,Y 178.402,Z 913.072,A -85,B 0,C 180,E1 -22638.461,E2 -22638.461} C_VEL
LIN {X 0,Y 178.422,Z 913.07,A -85,B 0,C 180,E1 -22643.782,E2 -22643.782} C_VEL
LIN {X 0,Y 178.487,Z 913.065,A -85,B 0,C 180,E1 -22646.545,E2 -22646.545} C_VEL
LIN {X 0,Y 178.442,Z 913.066,A -85,B 0,C 180,E1 -22651.794,E2 -22651.794} C_VEL
LIN {X 0,Y 178.466,Z 913.067,A -85,B 0,C 180,E1 -22656.808,E2 -22656.808} C_VEL
LIN {X 0,Y 178.608,Z 913.048,A -85,B 0,C 180,E1 -22661.651,E2 -22661.651} C_VEL
LIN {X 0,Y 178.634,Z 913.042,A -85,B 0,C 180,E1 -22666.345,E2 -22666.345} C_VEL
LIN {X 0,Y 178.908,Z 913.009,A -85,B 0,C 180,E1 -22670.958,E2 -22670.958} C_VEL
LIN {X 0,Y 178.82,Z 913.022,A -85,B 0,C 180,E1 -22675.491,E2 -22675.491} C_VEL
LIN {X 0,Y 179.342,Z 912.957,A -85,B 0,C 180,E1 -22679.999,E2 -22679.999} C_VEL
LIN {X 0,Y 178.893,Z 913.008,A -85,B 0,C 180,E1 -22686.767,E2 -22686.767} C_VEL
LIN {X 0,Y 178.835,Z 913.021,A -85,B 0,C 180,E1 -22690.74,E2 -22690.74} C_VEL
LIN {X 0,Y 178.577,Z 913.047,A -85,B 0,C 180,E1 -22695.99,E2 -22695.99} C_VEL
LIN {X 0,Y 178.555,Z 913.056,A -85,B 0,C 180,E1 -22699.151,E2 -22699.151} C_VEL
LIN {X 0,Y 178.465,Z 913.062,A -85,B 0,C 180,E1 -22705.075,E2 -22705.075} C_VEL
LIN {X 0,Y 178.46,Z 913.067,A -85,B 0,C 180,E1 -22710.793,E2 -22710.793} C_VEL
LIN {X 0,Y 178.483,Z 913.057,A -85,B 0,C 180,E1 -22714.217,E2 -22714.217} C_VEL
LIN {X 0,Y 178.387,Z 913.075,A -85,B 0,C 180,E1 -22719.075,E2 -22719.075} C_VEL
LIN {X 0,Y 178.393,Z 913.073,A -85,B 0,C 180,E1 -22722.045,E2 -22722.045} C_VEL
LIN {X 0,Y 178.391,Z 913.071,A -85,B 0,C 180,E1 -22725.164,E2 -22725.164} C_VEL
LIN {X 0,Y 178.397,Z 913.075,A -85,B 0,C 180,E1 -22728.46,E2 -22728.46} C_VEL
LIN {X 0,Y 178.418,Z 913.066,A -85,B 0,C 180,E1 -22733.781,E2 -22733.781} C_VEL
LIN {X 0,Y 178.568,Z 913.052,A -85,B 0,C 180,E1 -22739.226,E2 -22739.226} C_VEL
LIN {X 0,Y 179.096,Z 913.125,A -85,B 0,C 180,E1 -22743.482,E2 -22743.482} C_VEL
LIN {X 0,Y 179.893,Z 917.146,A -85,B 0,C 180,E1 -22745.781,E2 -22745.781} C_VEL
LIN {X 0,Y 179.071,Z 921.919,A -85,B 0,C 180,E1 -22748.486,E2 -22748.486} C_VEL
LIN {X 0,Y 179.487,Z 940.237,A -85,B 0,C 180,E1 -22749.818,E2 -22749.818} C_VEL
LIN {X 0,Y 181.716,Z 966.753,A -85,B 0,C 180,E1 -22751.703,E2 -22751.703} C_VEL
LIN {X 0,Y 180.754,Z 1001.748,A -85,B 0,C 180,E1 -22754.351,E2 -22754.351} C_VEL
LIN {X 0,Y 180.054,Z 1013.754,A -85,B 0,C 180,E1 -22755.735,E2 -22755.735} C_VEL
LIN {X 0,Y 179.609,Z 1023.819,A -85,B 0,C 180,E1 -22757.284,E2 -22757.284} C_VEL
LIN {X 0,Y 178.923,Z 1034.806,A -85,B 0,C 180,E1 -22759.451,E2 -22759.451} C_VEL
LIN {X 0,Y 178.475,Z 1042.967,A -85,B 0,C 180,E1 -22761.508,E2 -22761.508} C_VEL
LIN {X 0,Y 178.185,Z 1050.371,A -85,B 0,C 180,E1 -22763.773,E2 -22763.773} C_VEL
LIN {X 0,Y 177.996,Z 1056.508,A -85,B 0,C 180,E1 -22766.037,E2 -22766.037} C_VEL
LIN {X 0,Y 177.771,Z 1061.545,A -85,B 0,C 180,E1 -22768.3,E2 -22768.3} C_VEL
LIN {X 0,Y 177.493,Z 1066.528,A -85,B 0,C 180,E1 -22771.134,E2 -22771.134} C_VEL
LIN {X 0,Y 177.01,Z 1071.035,A -85,B 0,C 180,E1 -22774.554,E2 -22774.554} C_VEL
LIN {X 0,Y 176.93,Z 1071.85,A -85,B 0,C 180,E1 -22775.27,E2 -22775.27} C_VEL
LIN {X 0,Y 176.219,Z 1073.573,A -85,B 0,C 180,E1 -22777.089,E2 -22777.089} C_VEL
LIN {X 0,Y 173.798,Z 1075.298,A -85,B 0,C 180,E1 -22780.189,E2 -22780.189} C_VEL
LIN {X 0,Y 172.214,Z 1076.088,A -85,B 0,C 180,E1 -22782.764,E2 -22782.764} C_VEL
LIN {X 0,Y 172.088,Z 1076.603,A -85,B 0,C 180,E1 -22784.731,E2 -22784.731} C_VEL
LIN {X 0,Y 172.36,Z 1076.776,A -85,B 0,C 180,E1 -22785.38,E2 -22785.38} C_VEL
LIN {X 0,Y 174.797,Z 1077.309,A -85,B 0,C 180,E1 -22788.763,E2 -22788.763} C_VEL
LIN {X 0,Y 176.805,Z 1077.153,A -85,B 0,C 180,E1 -22790.962,E2 -22790.962} C_VEL
LIN {X 0,Y 179.198,Z 1076.598,A -85,B 0,C 180,E1 -22793.091,E2 -22793.091} C_VEL
LIN {X 0,Y 181.925,Z 1075.503,A -85,B 0,C 180,E1 -22795.147,E2 -22795.147} C_VEL
LIN {X 0,Y 188.502,Z 1072.171,A -85,B 0,C 180,E1 -22798.991,E2 -22798.991} C_VEL
LIN {X 0,Y 194.16,Z 1068.324,A -85,B 0,C 180,E1 -22801.658,E2 -22801.658} C_VEL
LIN {X 0,Y 200.456,Z 1063.315,A -85,B 0,C 180,E1 -22804.122,E2 -22804.122} C_VEL
LIN {X 0,Y 206.113,Z 1058.104,A -85,B 0,C 180,E1 -22806.028,E2 -22806.028} C_VEL
LIN {X 0,Y 212.2,Z 1051.824,A -85,B 0,C 180,E1 -22807.786,E2 -22807.786} C_VEL
LIN {X 0,Y 218.442,Z 1044.493,A -85,B 0,C 180,E1 -22809.335,E2 -22809.335} C_VEL
LIN {X 0,Y 225.552,Z 1034.747,A -85,B 0,C 180,E1 -22810.869,E2 -22810.869} C_VEL
LIN {X 0,Y 231.283,Z 1025.482,A -85,B 0,C 180,E1 -22811.952,E2 -22811.952} C_VEL
LIN {X 0,Y 236.321,Z 1015.838,A -85,B 0,C 180,E1 -22812.832,E2 -22812.832} C_VEL
LIN {X 0,Y 240.582,Z 1006.268,A -85,B 0,C 180,E1 -22813.496,E2 -22813.496} C_VEL
LIN {X 0,Y 241.139,Z 1004.317,A -85,B 0,C 180,E1 -22814.385,E2 -22814.385} C_VEL
LIN {X 0,Y 241.227,Z 1003.593,A -85,B 0,C 180,E1 -22815.636,E2 -22815.636} C_VEL
LIN {X 0,Y 241.405,Z 1003.57,A -85,B 0,C 180,E1 -22817.054,E2 -22817.054} C_VEL
LIN {X 0,Y 240.476,Z 1005.865,A -85,B 0,C 180,E1 -22817.308,E2 -22817.308} C_VEL
LIN {X 0,Y 235.921,Z 1015.746,A -85,B 0,C 180,E1 -22818.172,E2 -22818.172} C_VEL
LIN {X 0,Y 230.489,Z 1025.704,A -85,B 0,C 180,E1 -22819.326,E2 -22819.326} C_VEL
LIN {X 0,Y 224.494,Z 1034.654,A -85,B 0,C 180,E1 -22820.659,E2 -22820.659} C_VEL
LIN {X 0,Y 218.193,Z 1042.732,A -85,B 0,C 180,E1 -22822.267,E2 -22822.267} C_VEL
LIN {X 0,Y 212.141,Z 1049.349,A -85,B 0,C 180,E1 -22823.983,E2 -22823.983} C_VEL
LIN {X 0,Y 206.406,Z 1054.8,A -85,B 0,C 180,E1 -22825.82,E2 -22825.82} C_VEL
LIN {X 0,Y 200.008,Z 1059.961,A -85,B 0,C 180,E1 -22828.193,E2 -22828.193} C_VEL
LIN {X 0,Y 194.011,Z 1063.805,A -85,B 0,C 180,E1 -22830.724,E2 -22830.724} C_VEL
LIN {X 0,Y 188.035,Z 1066.728,A -85,B 0,C 180,E1 -22833.769,E2 -22833.769} C_VEL
LIN {X 0,Y 185.307,Z 1067.754,A -85,B 0,C 180,E1 -22835.344,E2 -22835.344} C_VEL
LIN {X 0,Y 182.266,Z 1068.5,A -85,B 0,C 180,E1 -22837.321,E2 -22837.321} C_VEL
LIN {X 0,Y 179.504,Z 1068.743,A -85,B 0,C 180,E1 -22839.369,E2 -22839.369} C_VEL
LIN {X 0,Y 177.119,Z 1068.592,A -85,B 0,C 180,E1 -22841.493,E2 -22841.493} C_VEL
LIN {X 0,Y 175.144,Z 1068.026,A -85,B 0,C 180,E1 -22843.688,E2 -22843.688} C_VEL
LIN {X 0,Y 173.489,Z 1066.901,A -85,B 0,C 180,E1 -22845.934,E2 -22845.934} C_VEL
LIN {X 0,Y 170.903,Z 1063.406,A -85,B 0,C 180,E1 -22850.533,E2 -22850.533} C_VEL
LIN {X 0,Y 170.021,Z 1059.843,A -85,B 0,C 180,E1 -22853.748,E2 -22853.748} C_VEL
LIN {X 0,Y 169.713,Z 1054.246,A -85,B 0,C 180,E1 -22857.628,E2 -22857.628} C_VEL
LIN {X 0,Y 169.768,Z 1048.794,A -85,B 0,C 180,E1 -22860.594,E2 -22860.594} C_VEL
LIN {X 0,Y 169.963,Z 1042.017,A -85,B 0,C 180,E1 -22863.557,E2 -22863.557} C_VEL
LIN {X 0,Y 170.447,Z 1033.566,A -85,B 0,C 180,E1 -22866.512,E2 -22866.512} C_VEL
LIN {X 0,Y 171.018,Z 1024.465,A -85,B 0,C 180,E1 -22869.066,E2 -22869.066} C_VEL
LIN {X 0,Y 171.642,Z 1015.333,A -85,B 0,C 180,E1 -22871.156,E2 -22871.156} C_VEL
LIN {X 0,Y 172.44,Z 1003.419,A -85,B 0,C 180,E1 -22873.254,E2 -22873.254} C_VEL
LIN {X 0,Y 173.015,Z 993.736,A -85,B 0,C 180,E1 -22874.558,E2 -22874.558} C_VEL
LIN {X 0,Y 173.392,Z 983.781,A -85,B 0,C 180,E1 -22875.578,E2 -22875.578} C_VEL
LIN {X 0,Y 174.712,Z 945.835,A -85,B 0,C 180,E1 -22878.546,E2 -22878.546} C_VEL
LIN {X 0,Y 175.044,Z 935.003,A -85,B 0,C 180,E1 -22879.37,E2 -22879.37} C_VEL
LIN {X 0,Y 172.665,Z 918.413,A -85,B 0,C 180,E1 -22880.583,E2 -22880.583} C_VEL
LIN {X 0,Y 171.797,Z 913.884,A -85,B 0,C 180,E1 -22880.965,E2 -22880.965} C_VEL
LIN {X 0,Y 171.391,Z 913.948,A -85,B 0,C 180,E1 -22886.813,E2 -22886.813} C_VEL
LIN {X 0,Y 171.41,Z 913.943,A -85,B 0,C 180,E1 -22892.211,E2 -22892.211} C_VEL
LIN {X 0,Y 171.393,Z 913.947,A -85,B 0,C 180,E1 -22895.036,E2 -22895.036} C_VEL
LIN {X 0,Y 171.344,Z 913.947,A -85,B 0,C 180,E1 -22898.802,E2 -22898.802} C_VEL
LIN {X 0,Y 171.32,Z 913.957,A -85,B 0,C 180,E1 -22904.219,E2 -22904.219} C_VEL
LIN {X 0,Y 171.332,Z 913.949,A -85,B 0,C 180,E1 -22908.981,E2 -22908.981} C_VEL
LIN {X 0,Y 171.362,Z 913.951,A -85,B 0,C 180,E1 -22912.035,E2 -22912.035} C_VEL
LIN {X 0,Y 171.4,Z 913.944,A -85,B 0,C 180,E1 -22915.094,E2 -22915.094} C_VEL
LIN {X 0,Y 171.412,Z 913.944,A -85,B 0,C 180,E1 -22920.528,E2 -22920.528} C_VEL
LIN {X 0,Y 171.44,Z 913.937,A -85,B 0,C 180,E1 -22925.799,E2 -22925.799} C_VEL
LIN {X 0,Y 171.511,Z 913.933,A -85,B 0,C 180,E1 -22930.864,E2 -22930.864} C_VEL
LIN {X 0,Y 171.56,Z 913.921,A -85,B 0,C 180,E1 -22935.772,E2 -22935.772} C_VEL
LIN {X 0,Y 171.848,Z 913.89,A -85,B 0,C 180,E1 -22940.585,E2 -22940.585} C_VEL
LIN {X 0,Y 171.773,Z 913.895,A -85,B 0,C 180,E1 -22945.307,E2 -22945.307} C_VEL
LIN {X 0,Y 172.309,Z 913.836,A -85,B 0,C 180,E1 -22950,E2 -22950} C_VEL
LIN {X 0,Y 171.861,Z 913.887,A -85,B 0,C 180,E1 -22957.047,E2 -22957.047} C_VEL
LIN {X 0,Y 171.771,Z 913.899,A -85,B 0,C 180,E1 -22960.893,E2 -22960.893} C_VEL
LIN {X 0,Y 171.509,Z 913.933,A -85,B 0,C 180,E1 -22966.67,E2 -22966.67} C_VEL
LIN {X 0,Y 171.482,Z 913.935,A -85,B 0,C 180,E1 -22969.499,E2 -22969.499} C_VEL
LIN {X 0,Y 171.407,Z 913.945,A -85,B 0,C 180,E1 -22975.57,E2 -22975.57} C_VEL
LIN {X 0,Y 171.422,Z 913.941,A -85,B 0,C 180,E1 -22980.572,E2 -22980.572} C_VEL
LIN {X 0,Y 171.396,Z 913.945,A -85,B 0,C 180,E1 -22985.035,E2 -22985.035} C_VEL
LIN {X 0,Y 171.347,Z 913.951,A -85,B 0,C 180,E1 -22988.801,E2 -22988.801} C_VEL
LIN {X 0,Y 171.323,Z 913.957,A -85,B 0,C 180,E1 -22994.218,E2 -22994.218} C_VEL
LIN {X 0,Y 171.334,Z 913.951,A -85,B 0,C 180,E1 -22998.979,E2 -22998.979} C_VEL
LIN {X 0,Y 171.364,Z 913.947,A -85,B 0,C 180,E1 -23002.033,E2 -23002.033} C_VEL
LIN {X 0,Y 171.401,Z 913.946,A -85,B 0,C 180,E1 -23005.092,E2 -23005.092} C_VEL
LIN {X 0,Y 171.411,Z 913.94,A -85,B 0,C 180,E1 -23010.526,E2 -23010.526} C_VEL
LIN {X 0,Y 171.406,Z 913.944,A -85,B 0,C 180,E1 -23015.793,E2 -23015.793} C_VEL
LIN {X 0,Y 171.511,Z 913.929,A -85,B 0,C 180,E1 -23020.863,E2 -23020.863} C_VEL
LIN {X 0,Y 171.549,Z 913.926,A -85,B 0,C 180,E1 -23025.769,E2 -23025.769} C_VEL
LIN {X 0,Y 171.846,Z 913.888,A -85,B 0,C 180,E1 -23030.584,E2 -23030.584} C_VEL
LIN {X 0,Y 171.771,Z 913.899,A -85,B 0,C 180,E1 -23035.305,E2 -23035.305} C_VEL
LIN {X 0,Y 172.307,Z 913.833,A -85,B 0,C 180,E1 -23039.999,E2 -23039.999} C_VEL
LIN {X 0,Y 171.856,Z 913.883,A -85,B 0,C 180,E1 -23047.046,E2 -23047.046} C_VEL
LIN {X 0,Y 171.768,Z 913.901,A -85,B 0,C 180,E1 -23050.892,E2 -23050.892} C_VEL
LIN {X 0,Y 171.51,Z 913.928,A -85,B 0,C 180,E1 -23056.668,E2 -23056.668} C_VEL
LIN {X 0,Y 171.479,Z 913.936,A -85,B 0,C 180,E1 -23059.497,E2 -23059.497} C_VEL
LIN {X 0,Y 171.403,Z 913.942,A -85,B 0,C 180,E1 -23065.568,E2 -23065.568} C_VEL
LIN {X 0,Y 171.418,Z 913.943,A -85,B 0,C 180,E1 -23070.571,E2 -23070.571} C_VEL
LIN {X 0,Y 171.392,Z 913.941,A -85,B 0,C 180,E1 -23075.034,E2 -23075.034} C_VEL
LIN {X 0,Y 171.343,Z 913.953,A -85,B 0,C 180,E1 -23078.8,E2 -23078.8} C_VEL
LIN {X 0,Y 171.318,Z 913.953,A -85,B 0,C 180,E1 -23084.217,E2 -23084.217} C_VEL
LIN {X 0,Y 171.329,Z 913.954,A -85,B 0,C 180,E1 -23088.979,E2 -23088.979} C_VEL
LIN {X 0,Y 171.359,Z 913.949,A -85,B 0,C 180,E1 -23092.033,E2 -23092.033} C_VEL
LIN {X 0,Y 171.397,Z 913.945,A -85,B 0,C 180,E1 -23095.092,E2 -23095.092} C_VEL
LIN {X 0,Y 171.638,Z 913.915,A -85,B 0,C 180,E1 -23100.569,E2 -23100.569} C_VEL
LIN {X 0,Y 172.133,Z 914.005,A -85,B 0,C 180,E1 -23103.925,E2 -23103.925} C_VEL
LIN {X 0,Y 172.74,Z 917.463,A -85,B 0,C 180,E1 -23105.992,E2 -23105.992} C_VEL
LIN {X 0,Y 171.984,Z 921.643,A -85,B 0,C 180,E1 -23108.469,E2 -23108.469} C_VEL
LIN {X 0,Y 172.351,Z 939.806,A -85,B 0,C 180,E1 -23109.855,E2 -23109.855} C_VEL
LIN {X 0,Y 174.621,Z 967.262,A -85,B 0,C 180,E1 -23111.901,E2 -23111.901} C_VEL
LIN {X 0,Y 173.769,Z 1000.858,A -85,B 0,C 180,E1 -23114.608,E2 -23114.608} C_VEL
LIN {X 0,Y 173.062,Z 1013.102,A -85,B 0,C 180,E1 -23116.062,E2 -23116.062} C_VEL
LIN {X 0,Y 172.698,Z 1022.104,A -85,B 0,C 180,E1 -23117.476,E2 -23117.476} C_VEL
LIN {X 0,Y 172.125,Z 1031.979,A -85,B 0,C 180,E1 -23119.432,E2 -23119.432} C_VEL
LIN {X 0,Y 171.603,Z 1041.382,A -85,B 0,C 180,E1 -23121.758,E2 -23121.758} C_VEL
LIN {X 0,Y 171.335,Z 1048.944,A -85,B 0,C 180,E1 -23124.114,E2 -23124.114} C_VEL
LIN {X 0,Y 171.144,Z 1055.14,A -85,B 0,C 180,E1 -23126.468,E2 -23126.468} C_VEL
LIN {X 0,Y 170.932,Z 1060.266,A -85,B 0,C 180,E1 -23128.822,E2 -23128.822} C_VEL
LIN {X 0,Y 170.657,Z 1064.5,A -85,B 0,C 180,E1 -23131.179,E2 -23131.179} C_VEL
LIN {X 0,Y 170.311,Z 1067.919,A -85,B 0,C 180,E1 -23133.548,E2 -23133.548} C_VEL
LIN {X 0,Y 170.026,Z 1071.952,A -85,B 0,C 180,E1 -23137.243,E2 -23137.243} C_VEL
LIN {X 0,Y 170.255,Z 1073.794,A -85,B 0,C 180,E1 -23139.504,E2 -23139.504} C_VEL
LIN {X 0,Y 170.779,Z 1075.306,A -85,B 0,C 180,E1 -23141.874,E2 -23141.874} C_VEL
LIN {X 0,Y 172.36,Z 1076.776,A -85,B 0,C 180,E1 -23145.38,E2 -23145.38} C_VEL
LIN {X 0,Y 172.935,Z 1077.195,A -85,B 0,C 180,E1 -23147.327,E2 -23147.327} C_VEL
LIN {X 0,Y 172.715,Z 1076.962,A -85,B 0,C 180,E1 -23151.926,E2 -23151.926} C_VEL
LIN {X 0,Y 173.678,Z 1076.35,A -85,B 0,C 180,E1 -23154.507,E2 -23154.507} C_VEL
LIN {X 0,Y 174.961,Z 1075.914,A -85,B 0,C 180,E1 -23155.72,E2 -23155.72} C_VEL
LIN {X 0,Y 178.795,Z 1074.62,A -85,B 0,C 180,E1 -23158.144,E2 -23158.144} C_VEL
LIN {X 0,Y 184.255,Z 1072.029,A -85,B 0,C 180,E1 -23160.992,E2 -23160.992} C_VEL
LIN {X 0,Y 190.357,Z 1068.399,A -85,B 0,C 180,E1 -23163.628,E2 -23163.628} C_VEL
LIN {X 0,Y 197.032,Z 1063.531,A -85,B 0,C 180,E1 -23166.053,E2 -23166.053} C_VEL
LIN {X 0,Y 204.235,Z 1057.426,A -85,B 0,C 180,E1 -23168.272,E2 -23168.272} C_VEL
LIN {X 0,Y 211.738,Z 1050.071,A -85,B 0,C 180,E1 -23170.152,E2 -23170.152} C_VEL
LIN {X 0,Y 219.118,Z 1041.641,A -85,B 0,C 180,E1 -23171.762,E2 -23171.762} C_VEL
LIN {X 0,Y 226.314,Z 1031.743,A -85,B 0,C 180,E1 -23173.093,E2 -23173.093} C_VEL
LIN {X 0,Y 232.341,Z 1022.165,A -85,B 0,C 180,E1 -23174.084,E2 -23174.084} C_VEL
LIN {X 0,Y 237.852,Z 1011.464,A -85,B 0,C 180,E1 -23174.903,E2 -23174.903} C_VEL
LIN {X 0,Y 238.272,Z 1010.467,A -85,B 0,C 180,E1 -23175.064,E2 -23175.064} C_VEL
LIN {X 0,Y 237.999,Z 1010.968,A -85,B 0,C 180,E1 -23175.934,E2 -23175.934} C_VEL
LIN {X 0,Y 232.705,Z 1021.086,A -85,B 0,C 180,E1 -23176.899,E2 -23176.899} C_VEL
LIN {X 0,Y 226.926,Z 1030.047,A -85,B 0,C 180,E1 -23178.012,E2 -23178.012} C_VEL
LIN {X 0,Y 220.911,Z 1038.16,A -85,B 0,C 180,E1 -23179.295,E2 -23179.295} C_VEL
LIN {X 0,Y 213.039,Z 1046.991,A -85,B 0,C 180,E1 -23181.187,E2 -23181.187} C_VEL
LIN {X 0,Y 206.828,Z 1052.87,A -85,B 0,C 180,E1 -23182.906,E2 -23182.906} C_VEL
LIN {X 0,Y 200.874,Z 1057.673,A -85,B 0,C 180,E1 -23184.741,E2 -23184.741} C_VEL
LIN {X 0,Y 194.213,Z 1062.201,A -85,B 0,C 180,E1 -23187.126,E2 -23187.126} C_VEL
LIN {X 0,Y 189.986,Z 1064.574,A -85,B 0,C 180,E1 -23188.81,E2 -23188.81} C_VEL
LIN {X 0,Y 186.075,Z 1066.451,A -85,B 0,C 180,E1 -23190.594,E2 -23190.594} C_VEL
LIN {X 0,Y 181.369,Z 1068.15,A -85,B 0,C 180,E1 -23193.029,E2 -23193.029} C_VEL
LIN {X 0,Y 175.781,Z 1069.153,A -85,B 0,C 180,E1 -23196.434,E2 -23196.434} C_VEL
LIN {X 0,Y 172.895,Z 1069.219,A -85,B 0,C 180,E1 -23198.542,E2 -23198.542} C_VEL
LIN {X 0,Y 170.426,Z 1068.72,A -85,B 0,C 180,E1 -23200.738,E2 -23200.738} C_VEL
LIN {X 0,Y 166.638,Z 1066.578,A -85,B 0,C 180,E1 -23205.343,E2 -23205.343} C_VEL
LIN {X 0,Y 164.506,Z 1063.686,A -85,B 0,C 180,E1 -23208.917,E2 -23208.917} C_VEL
LIN {X 0,Y 163.217,Z 1059.736,A -85,B 0,C 180,E1 -23212.579,E2 -23212.579} C_VEL
LIN {X 0,Y 162.891,Z 1056.508,A -85,B 0,C 180,E1 -23215.051,E2 -23215.051} C_VEL
LIN {X 0,Y 162.771,Z 1051.509,A -85,B 0,C 180,E1 -23218.145,E2 -23218.145} C_VEL
LIN {X 0,Y 162.929,Z 1045.387,A -85,B 0,C 180,E1 -23221.237,E2 -23221.237} C_VEL
LIN {X 0,Y 163.114,Z 1039.484,A -85,B 0,C 180,E1 -23223.707,E2 -23223.707} C_VEL
LIN {X 0,Y 163.543,Z 1032.378,A -85,B 0,C 180,E1 -23226.169,E2 -23226.169} C_VEL
LIN {X 0,Y 164.057,Z 1023.551,A -85,B 0,C 180,E1 -23228.689,E2 -23228.689} C_VEL
LIN {X 0,Y 164.753,Z 1013.231,A -85,B 0,C 180,E1 -23231.07,E2 -23231.07} C_VEL
LIN {X 0,Y 165.435,Z 1003.064,A -85,B 0,C 180,E1 -23232.888,E2 -23232.888} C_VEL
LIN {X 0,Y 165.987,Z 993.448,A -85,B 0,C 180,E1 -23234.248,E2 -23234.248} C_VEL
LIN {X 0,Y 166.343,Z 982.732,A -85,B 0,C 180,E1 -23235.391,E2 -23235.391} C_VEL
LIN {X 0,Y 167.633,Z 945.85,A -85,B 0,C 180,E1 -23238.407,E2 -23238.407} C_VEL
LIN {X 0,Y 167.874,Z 934.846,A -85,B 0,C 180,E1 -23239.28,E2 -23239.28} C_VEL
LIN {X 0,Y 165.707,Z 919.753,A -85,B 0,C 180,E1 -23240.432,E2 -23240.432} C_VEL
LIN {X 0,Y 164.77,Z 914.76,A -85,B 0,C 180,E1 -23240.821,E2 -23240.821} C_VEL
LIN {X 0,Y 164.371,Z 914.821,A -85,B 0,C 180,E1 -23246.118,E2 -23246.118} C_VEL
LIN {X 0,Y 164.359,Z 914.819,A -85,B 0,C 180,E1 -23251.218,E2 -23251.218} C_VEL
LIN {X 0,Y 164.281,Z 914.831,A -85,B 0,C 180,E1 -23256.795,E2 -23256.795} C_VEL
LIN {X 0,Y 164.287,Z 914.828,A -85,B 0,C 180,E1 -23259.919,E2 -23259.919} C_VEL
LIN {X 0,Y 164.282,Z 914.833,A -85,B 0,C 180,E1 -23263.343,E2 -23263.343} C_VEL
LIN {X 0,Y 164.263,Z 914.832,A -85,B 0,C 180,E1 -23266.799,E2 -23266.799} C_VEL
LIN {X 0,Y 164.291,Z 914.831,A -85,B 0,C 180,E1 -23270.356,E2 -23270.356} C_VEL
LIN {X 0,Y 164.328,Z 914.829,A -85,B 0,C 180,E1 -23274.352,E2 -23274.352} C_VEL
LIN {X 0,Y 164.37,Z 914.82,A -85,B 0,C 180,E1 -23279.131,E2 -23279.131} C_VEL
LIN {X 0,Y 164.397,Z 914.818,A -85,B 0,C 180,E1 -23284.691,E2 -23284.691} C_VEL
LIN {X 0,Y 164.42,Z 914.814,A -85,B 0,C 180,E1 -23290.118,E2 -23290.118} C_VEL
LIN {X 0,Y 164.488,Z 914.804,A -85,B 0,C 180,E1 -23295.146,E2 -23295.146} C_VEL
LIN {X 0,Y 164.769,Z 914.772,A -85,B 0,C 180,E1 -23300.177,E2 -23300.177} C_VEL
LIN {X 0,Y 164.823,Z 914.764,A -85,B 0,C 180,E1 -23302.651,E2 -23302.651} C_VEL
LIN {X 0,Y 165.273,Z 914.712,A -85,B 0,C 180,E1 -23310,E2 -23310} C_VEL
LIN {X 0,Y 164.823,Z 914.764,A -85,B 0,C 180,E1 -23317.35,E2 -23317.35} C_VEL
LIN {X 0,Y 164.706,Z 914.778,A -85,B 0,C 180,E1 -23321.058,E2 -23321.058} C_VEL
LIN {X 0,Y 164.432,Z 914.814,A -85,B 0,C 180,E1 -23327.409,E2 -23327.409} C_VEL
LIN {X 0,Y 164.423,Z 914.814,A -85,B 0,C 180,E1 -23329.996,E2 -23329.996} C_VEL
LIN {X 0,Y 164.343,Z 914.824,A -85,B 0,C 180,E1 -23336.094,E2 -23336.094} C_VEL
LIN {X 0,Y 164.357,Z 914.82,A -85,B 0,C 180,E1 -23341.214,E2 -23341.214} C_VEL
LIN {X 0,Y 164.284,Z 914.832,A -85,B 0,C 180,E1 -23346.793,E2 -23346.793} C_VEL
LIN {X 0,Y 164.29,Z 914.829,A -85,B 0,C 180,E1 -23349.917,E2 -23349.917} C_VEL
LIN {X 0,Y 164.284,Z 914.829,A -85,B 0,C 180,E1 -23353.341,E2 -23353.341} C_VEL
LIN {X 0,Y 164.265,Z 914.834,A -85,B 0,C 180,E1 -23356.798,E2 -23356.798} C_VEL
LIN {X 0,Y 164.293,Z 914.827,A -85,B 0,C 180,E1 -23360.354,E2 -23360.354} C_VEL
LIN {X 0,Y 164.329,Z 914.828,A -85,B 0,C 180,E1 -23364.351,E2 -23364.351} C_VEL
LIN {X 0,Y 164.374,Z 914.816,A -85,B 0,C 180,E1 -23369.13,E2 -23369.13} C_VEL
LIN {X 0,Y 164.361,Z 914.825,A -85,B 0,C 180,E1 -23374.684,E2 -23374.684} C_VEL
LIN {X 0,Y 164.419,Z 914.811,A -85,B 0,C 180,E1 -23380.117,E2 -23380.117} C_VEL
LIN {X 0,Y 164.479,Z 914.81,A -85,B 0,C 180,E1 -23385.144,E2 -23385.144} C_VEL
LIN {X 0,Y 164.768,Z 914.77,A -85,B 0,C 180,E1 -23390.175,E2 -23390.175} C_VEL
LIN {X 0,Y 164.821,Z 914.765,A -85,B 0,C 180,E1 -23392.649,E2 -23392.649} C_VEL
LIN {X 0,Y 165.271,Z 914.709,A -85,B 0,C 180,E1 -23399.999,E2 -23399.999} C_VEL
LIN {X 0,Y 164.818,Z 914.76,A -85,B 0,C 180,E1 -23407.348,E2 -23407.348} C_VEL
LIN {X 0,Y 164.703,Z 914.781,A -85,B 0,C 180,E1 -23411.056,E2 -23411.056} C_VEL
LIN {X 0,Y 164.432,Z 914.811,A -85,B 0,C 180,E1 -23417.408,E2 -23417.408} C_VEL
LIN {X 0,Y 164.42,Z 914.815,A -85,B 0,C 180,E1 -23419.995,E2 -23419.995} C_VEL
LIN {X 0,Y 164.339,Z 914.82,A -85,B 0,C 180,E1 -23426.093,E2 -23426.093} C_VEL
LIN {X 0,Y 164.357,Z 914.825,A -85,B 0,C 180,E1 -23431.216,E2 -23431.216} C_VEL
LIN {X 0,Y 164.279,Z 914.831,A -85,B 0,C 180,E1 -23436.792,E2 -23436.792} C_VEL
LIN {X 0,Y 164.285,Z 914.834,A -85,B 0,C 180,E1 -23439.917,E2 -23439.917} C_VEL
LIN {X 0,Y 164.279,Z 914.829,A -85,B 0,C 180,E1 -23443.341,E2 -23443.341} C_VEL
LIN {X 0,Y 164.26,Z 914.835,A -85,B 0,C 180,E1 -23446.797,E2 -23446.797} C_VEL
LIN {X 0,Y 164.288,Z 914.832,A -85,B 0,C 180,E1 -23450.354,E2 -23450.354} C_VEL
LIN {X 0,Y 164.338,Z 914.826,A -85,B 0,C 180,E1 -23456.223,E2 -23456.223} C_VEL
LIN {X 0,Y 164.963,Z 914.747,A -85,B 0,C 180,E1 -23463.464,E2 -23463.464} C_VEL
LIN {X 0,Y 165.226,Z 914.963,A -85,B 0,C 180,E1 -23464.498,E2 -23464.498} C_VEL
LIN {X 0,Y 165.562,Z 917.726,A -85,B 0,C 180,E1 -23466.217,E2 -23466.217} C_VEL
LIN {X 0,Y 164.914,Z 921.55,A -85,B 0,C 180,E1 -23468.535,E2 -23468.535} C_VEL
LIN {X 0,Y 165.272,Z 939.762,A -85,B 0,C 180,E1 -23469.987,E2 -23469.987} C_VEL
LIN {X 0,Y 167.554,Z 967.377,A -85,B 0,C 180,E1 -23472.138,E2 -23472.138} C_VEL
LIN {X 0,Y 166.743,Z 1000.681,A -85,B 0,C 180,E1 -23474.96,E2 -23474.96} C_VEL
LIN {X 0,Y 166.093,Z 1013.295,A -85,B 0,C 180,E1 -23476.543,E2 -23476.543} C_VEL
LIN {X 0,Y 165.662,Z 1022.549,A -85,B 0,C 180,E1 -23478.1,E2 -23478.1} C_VEL
LIN {X 0,Y 165.136,Z 1032.393,A -85,B 0,C 180,E1 -23480.198,E2 -23480.198} C_VEL
LIN {X 0,Y 164.715,Z 1041.567,A -85,B 0,C 180,E1 -23482.645,E2 -23482.645} C_VEL
LIN {X 0,Y 164.475,Z 1048.939,A -85,B 0,C 180,E1 -23485.097,E2 -23485.097} C_VEL
LIN {X 0,Y 164.295,Z 1055.038,A -85,B 0,C 180,E1 -23487.548,E2 -23487.548} C_VEL
LIN {X 0,Y 164.048,Z 1060.067,A -85,B 0,C 180,E1 -23490,E2 -23490} C_VEL
LIN {X 0,Y 163.722,Z 1064.134,A -85,B 0,C 180,E1 -23492.46,E2 -23492.46} C_VEL
LIN {X 0,Y 163.214,Z 1069.163,A -85,B 0,C 180,E1 -23496.529,E2 -23496.529} C_VEL
LIN {X 0,Y 163.423,Z 1072.315,A -85,B 0,C 180,E1 -23499.905,E2 -23499.905} C_VEL
LIN {X 0,Y 163.925,Z 1074.1,A -85,B 0,C 180,E1 -23502.378,E2 -23502.378} C_VEL
LIN {X 0,Y 165.496,Z 1075.771,A -85,B 0,C 180,E1 -23505.872,E2 -23505.872} C_VEL
LIN {X 0,Y 168.111,Z 1076.803,A -85,B 0,C 180,E1 -23509.538,E2 -23509.538} C_VEL
LIN {X 0,Y 170.195,Z 1076.863,A -85,B 0,C 180,E1 -23511.817,E2 -23511.817} C_VEL
LIN {X 0,Y 174.961,Z 1075.914,A -85,B 0,C 180,E1 -23515.72,E2 -23515.72} C_VEL
LIN {X 0,Y 176.932,Z 1075.214,A -85,B 0,C 180,E1 -23517.522,E2 -23517.522} C_VEL
LIN {X 0,Y 179.134,Z 1073.563,A -85,B 0,C 180,E1 -23520.59,E2 -23520.59} C_VEL
LIN {X 0,Y 182,Z 1071.276,A -85,B 0,C 180,E1 -23523.486,E2 -23523.486} C_VEL
LIN {X 0,Y 184.912,Z 1069.474,A -85,B 0,C 180,E1 -23524.975,E2 -23524.975} C_VEL
LIN {X 0,Y 191.465,Z 1065.497,A -85,B 0,C 180,E1 -23527.276,E2 -23527.276} C_VEL
LIN {X 0,Y 200.163,Z 1059.109,A -85,B 0,C 180,E1 -23529.85,E2 -23529.85} C_VEL
LIN {X 0,Y 207.492,Z 1052.695,A -85,B 0,C 180,E1 -23531.596,E2 -23531.596} C_VEL
LIN {X 0,Y 215.441,Z 1044.515,A -85,B 0,C 180,E1 -23533.239,E2 -23533.239} C_VEL
LIN {X 0,Y 222.971,Z 1035.555,A -85,B 0,C 180,E1 -23534.532,E2 -23534.532} C_VEL
LIN {X 0,Y 227.594,Z 1029.046,A -85,B 0,C 180,E1 -23535.253,E2 -23535.253} C_VEL
LIN {X 0,Y 228.477,Z 1027.708,A -85,B 0,C 180,E1 -23535.772,E2 -23535.772} C_VEL
LIN {X 0,Y 221.201,Z 1037.285,A -85,B 0,C 180,E1 -23537.116,E2 -23537.116} C_VEL
LIN {X 0,Y 214.684,Z 1044.481,A -85,B 0,C 180,E1 -23538.478,E2 -23538.478} C_VEL
LIN {X 0,Y 207.982,Z 1050.953,A -85,B 0,C 180,E1 -23540.057,E2 -23540.057} C_VEL
LIN {X 0,Y 200.277,Z 1057.104,A -85,B 0,C 180,E1 -23542.114,E2 -23542.114} C_VEL
LIN {X 0,Y 193.032,Z 1061.857,A -85,B 0,C 180,E1 -23544.372,E2 -23544.372} C_VEL
LIN {X 0,Y 188.478,Z 1064.387,A -85,B 0,C 180,E1 -23545.992,E2 -23545.992} C_VEL
LIN {X 0,Y 184.099,Z 1066.371,A -85,B 0,C 180,E1 -23547.694,E2 -23547.694} C_VEL
LIN {X 0,Y 176.197,Z 1068.89,A -85,B 0,C 180,E1 -23551.404,E2 -23551.404} C_VEL
LIN {X 0,Y 172.611,Z 1069.556,A -85,B 0,C 180,E1 -23553.394,E2 -23553.394} C_VEL
LIN {X 0,Y 169.318,Z 1069.673,A -85,B 0,C 180,E1 -23555.477,E2 -23555.477} C_VEL
LIN {X 0,Y 166.31,Z 1069.378,A -85,B 0,C 180,E1 -23557.647,E2 -23557.647} C_VEL
LIN {X 0,Y 163.748,Z 1068.727,A -85,B 0,C 180,E1 -23559.92,E2 -23559.92} C_VEL
LIN {X 0,Y 161.587,Z 1067.57,A -85,B 0,C 180,E1 -23562.276,E2 -23562.276} C_VEL
LIN {X 0,Y 158.997,Z 1065.06,A -85,B 0,C 180,E1 -23565.931,E2 -23565.931} C_VEL
LIN {X 0,Y 156.874,Z 1060.801,A -85,B 0,C 180,E1 -23570.265,E2 -23570.265} C_VEL
LIN {X 0,Y 156.141,Z 1056.721,A -85,B 0,C 180,E1 -23573.54,E2 -23573.54} C_VEL
LIN {X 0,Y 155.916,Z 1051.839,A -85,B 0,C 180,E1 -23576.771,E2 -23576.771} C_VEL
LIN {X 0,Y 155.998,Z 1045.758,A -85,B 0,C 180,E1 -23580.001,E2 -23580.001} C_VEL
LIN {X 0,Y 156.182,Z 1039.904,A -85,B 0,C 180,E1 -23582.58,E2 -23582.58} C_VEL
LIN {X 0,Y 156.647,Z 1031.048,A -85,B 0,C 180,E1 -23585.795,E2 -23585.795} C_VEL
LIN {X 0,Y 157.173,Z 1021.828,A -85,B 0,C 180,E1 -23588.497,E2 -23588.497} C_VEL
LIN {X 0,Y 157.904,Z 1011.16,A -85,B 0,C 180,E1 -23590.906,E2 -23590.906} C_VEL
LIN {X 0,Y 158.594,Z 1000.534,A -85,B 0,C 180,E1 -23592.803,E2 -23592.803} C_VEL
LIN {X 0,Y 159.255,Z 988.081,A -85,B 0,C 180,E1 -23594.456,E2 -23594.456} C_VEL
LIN {X 0,Y 160.49,Z 947.348,A -85,B 0,C 180,E1 -23598.099,E2 -23598.099} C_VEL
LIN {X 0,Y 160.786,Z 935.138,A -85,B 0,C 180,E1 -23599.138,E2 -23599.138} C_VEL
LIN {X 0,Y 158.736,Z 920.915,A -85,B 0,C 180,E1 -23600.271,E2 -23600.271} C_VEL
LIN {X 0,Y 157.75,Z 915.635,A -85,B 0,C 180,E1 -23600.755,E2 -23600.755} C_VEL
LIN {X 0,Y 157.311,Z 915.701,A -85,B 0,C 180,E1 -23606.682,E2 -23606.682} C_VEL
LIN {X 0,Y 157.269,Z 915.704,A -85,B 0,C 180,E1 -23612.43,E2 -23612.43} C_VEL
LIN {X 0,Y 157.26,Z 915.706,A -85,B 0,C 180,E1 -23616.446,E2 -23616.446} C_VEL
LIN {X 0,Y 157.191,Z 915.717,A -85,B 0,C 180,E1 -23622.119,E2 -23622.119} C_VEL
LIN {X 0,Y 157.192,Z 915.712,A -85,B 0,C 180,E1 -23627.884,E2 -23627.884} C_VEL
LIN {X 0,Y 157.261,Z 915.707,A -85,B 0,C 180,E1 -23633.557,E2 -23633.557} C_VEL
LIN {X 0,Y 157.283,Z 915.698,A -85,B 0,C 180,E1 -23638.105,E2 -23638.105} C_VEL
LIN {X 0,Y 157.312,Z 915.7,A -85,B 0,C 180,E1 -23643.465,E2 -23643.465} C_VEL
LIN {X 0,Y 157.363,Z 915.694,A -85,B 0,C 180,E1 -23649.703,E2 -23649.703} C_VEL
LIN {X 0,Y 157.42,Z 915.685,A -85,B 0,C 180,E1 -23654.463,E2 -23654.463} C_VEL
LIN {X 0,Y 157.692,Z 915.655,A -85,B 0,C 180,E1 -23659.731,E2 -23659.731} C_VEL
LIN {X 0,Y 157.762,Z 915.644,A -85,B 0,C 180,E1 -23662.32,E2 -23662.32} C_VEL
LIN {X 0,Y 158.235,Z 915.589,A -85,B 0,C 180,E1 -23670,E2 -23670} C_VEL
LIN {X 0,Y 157.762,Z 915.644,A -85,B 0,C 180,E1 -23677.681,E2 -23677.681} C_VEL
LIN {X 0,Y 157.635,Z 915.659,A -85,B 0,C 180,E1 -23681.224,E2 -23681.224} C_VEL
LIN {X 0,Y 157.41,Z 915.686,A -85,B 0,C 180,E1 -23685.539,E2 -23685.539} C_VEL
LIN {X 0,Y 157.307,Z 915.7,A -85,B 0,C 180,E1 -23690.942,E2 -23690.942} C_VEL
LIN {X 0,Y 157.27,Z 915.706,A -85,B 0,C 180,E1 -23696.649,E2 -23696.649} C_VEL
LIN {X 0,Y 157.268,Z 915.699,A -85,B 0,C 180,E1 -23702.43,E2 -23702.43} C_VEL
LIN {X 0,Y 157.262,Z 915.707,A -85,B 0,C 180,E1 -23706.444,E2 -23706.444} C_VEL
LIN {X 0,Y 157.194,Z 915.712,A -85,B 0,C 180,E1 -23712.117,E2 -23712.117} C_VEL
LIN {X 0,Y 157.194,Z 915.717,A -85,B 0,C 180,E1 -23717.882,E2 -23717.882} C_VEL
LIN {X 0,Y 157.262,Z 915.706,A -85,B 0,C 180,E1 -23723.555,E2 -23723.555} C_VEL
LIN {X 0,Y 157.287,Z 915.703,A -85,B 0,C 180,E1 -23728.101,E2 -23728.101} C_VEL
LIN {X 0,Y 157.271,Z 915.706,A -85,B 0,C 180,E1 -23733.455,E2 -23733.455} C_VEL
LIN {X 0,Y 157.362,Z 915.69,A -85,B 0,C 180,E1 -23739.702,E2 -23739.702} C_VEL
LIN {X 0,Y 157.412,Z 915.688,A -85,B 0,C 180,E1 -23744.46,E2 -23744.46} C_VEL
LIN {X 0,Y 157.69,Z 915.651,A -85,B 0,C 180,E1 -23749.73,E2 -23749.73} C_VEL
LIN {X 0,Y 157.76,Z 915.645,A -85,B 0,C 180,E1 -23752.318,E2 -23752.318} C_VEL
LIN {X 0,Y 158.233,Z 915.585,A -85,B 0,C 180,E1 -23759.999,E2 -23759.999} C_VEL
LIN {X 0,Y 157.757,Z 915.64,A -85,B 0,C 180,E1 -23767.679,E2 -23767.679} C_VEL
LIN {X 0,Y 157.632,Z 915.661,A -85,B 0,C 180,E1 -23771.222,E2 -23771.222} C_VEL
LIN {X 0,Y 157.41,Z 915.683,A -85,B 0,C 180,E1 -23775.537,E2 -23775.537} C_VEL
LIN {X 0,Y 157.304,Z 915.704,A -85,B 0,C 180,E1 -23780.941,E2 -23780.941} C_VEL
LIN {X 0,Y 157.266,Z 915.702,A -85,B 0,C 180,E1 -23786.648,E2 -23786.648} C_VEL
LIN {X 0,Y 157.268,Z 915.704,A -85,B 0,C 180,E1 -23792.428,E2 -23792.428} C_VEL
LIN {X 0,Y 157.258,Z 915.705,A -85,B 0,C 180,E1 -23796.443,E2 -23796.443} C_VEL
LIN {X 0,Y 157.189,Z 915.713,A -85,B 0,C 180,E1 -23802.116,E2 -23802.116} C_VEL
LIN {X 0,Y 157.189,Z 915.717,A -85,B 0,C 180,E1 -23807.881,E2 -23807.881} C_VEL
LIN {X 0,Y 157.258,Z 915.701,A -85,B 0,C 180,E1 -23813.554,E2 -23813.554} C_VEL
LIN {X 0,Y 157.353,Z 915.696,A -85,B 0,C 180,E1 -23818.059,E2 -23818.059} C_VEL
LIN {X 0,Y 158.287,Z 915.755,A -85,B 0,C 180,E1 -23825.051,E2 -23825.051} C_VEL
LIN {X 0,Y 158.38,Z 917.914,A -85,B 0,C 180,E1 -23826.461,E2 -23826.461} C_VEL
LIN {X 0,Y 157.81,Z 921.082,A -85,B 0,C 180,E1 -23828.529,E2 -23828.529} C_VEL
LIN {X 0,Y 158.214,Z 940.124,A -85,B 0,C 180,E1 -23830.159,E2 -23830.159} C_VEL
LIN {X 0,Y 160.515,Z 967.476,A -85,B 0,C 180,E1 -23832.399,E2 -23832.399} C_VEL
LIN {X 0,Y 159.721,Z 1000.611,A -85,B 0,C 180,E1 -23835.407,E2 -23835.407} C_VEL
LIN {X 0,Y 159.168,Z 1012.438,A -85,B 0,C 180,E1 -23836.977,E2 -23836.977} C_VEL
LIN {X 0,Y 158.746,Z 1021.852,A -85,B 0,C 180,E1 -23838.636,E2 -23838.636} C_VEL
LIN {X 0,Y 158.276,Z 1031.362,A -85,B 0,C 180,E1 -23840.737,E2 -23840.737} C_VEL
LIN {X 0,Y 157.881,Z 1041.676,A -85,B 0,C 180,E1 -23843.61,E2 -23843.61} C_VEL
LIN {X 0,Y 157.653,Z 1048.918,A -85,B 0,C 180,E1 -23846.165,E2 -23846.165} C_VEL
LIN {X 0,Y 157.507,Z 1054.819,A -85,B 0,C 180,E1 -23848.721,E2 -23848.721} C_VEL
LIN {X 0,Y 157.23,Z 1059.662,A -85,B 0,C 180,E1 -23851.28,E2 -23851.28} C_VEL
LIN {X 0,Y 156.83,Z 1063.647,A -85,B 0,C 180,E1 -23853.854,E2 -23853.854} C_VEL
LIN {X 0,Y 156.415,Z 1068.235,A -85,B 0,C 180,E1 -23857.746,E2 -23857.746} C_VEL
LIN {X 0,Y 156.624,Z 1070.701,A -85,B 0,C 180,E1 -23860.339,E2 -23860.339} C_VEL
LIN {X 0,Y 158.163,Z 1074.167,A -85,B 0,C 180,E1 -23865.462,E2 -23865.462} C_VEL
LIN {X 0,Y 159.593,Z 1075.356,A -85,B 0,C 180,E1 -23867.954,E2 -23867.954} C_VEL
LIN {X 0,Y 163.637,Z 1076.353,A -85,B 0,C 180,E1 -23872.739,E2 -23872.739} C_VEL
LIN {X 0,Y 166.241,Z 1076.35,A -85,B 0,C 180,E1 -23875.009,E2 -23875.009} C_VEL
LIN {X 0,Y 169.208,Z 1075.824,A -85,B 0,C 180,E1 -23877.186,E2 -23877.186} C_VEL
LIN {X 0,Y 176.273,Z 1073.685,A -85,B 0,C 180,E1 -23881.218,E2 -23881.218} C_VEL
LIN {X 0,Y 182.369,Z 1070.881,A -85,B 0,C 180,E1 -23883.972,E2 -23883.972} C_VEL
LIN {X 0,Y 184.912,Z 1069.474,A -85,B 0,C 180,E1 -23884.975,E2 -23884.975} C_VEL
LIN {X 0,Y 188.039,Z 1067.622,A -85,B 0,C 180,E1 -23886.415,E2 -23886.415} C_VEL
LIN {X 0,Y 192.15,Z 1064.502,A -85,B 0,C 180,E1 -23888.98,E2 -23888.98} C_VEL
LIN {X 0,Y 196.569,Z 1060.709,A -85,B 0,C 180,E1 -23891.313,E2 -23891.313} C_VEL
LIN {X 0,Y 200.049,Z 1057.809,A -85,B 0,C 180,E1 -23892.379,E2 -23892.379} C_VEL
LIN {X 0,Y 207.609,Z 1051.484,A -85,B 0,C 180,E1 -23893.945,E2 -23893.945} C_VEL
LIN {X 0,Y 213.543,Z 1045.767,A -85,B 0,C 180,E1 -23895.039,E2 -23895.039} C_VEL
LIN {X 0,Y 216.591,Z 1042.541,A -85,B 0,C 180,E1 -23895.55,E2 -23895.55} C_VEL
LIN {X 0,Y 216.507,Z 1042.583,A -85,B 0,C 180,E1 -23895.959,E2 -23895.959} C_VEL
LIN {X 0,Y 210.052,Z 1048.783,A -85,B 0,C 180,E1 -23897.249,E2 -23897.249} C_VEL
LIN {X 0,Y 202.901,Z 1054.578,A -85,B 0,C 180,E1 -23898.845,E2 -23898.845} C_VEL
LIN {X 0,Y 194.982,Z 1060.054,A -85,B 0,C 180,E1 -23900.894,E2 -23900.894} C_VEL
LIN {X 0,Y 187.517,Z 1064.194,A -85,B 0,C 180,E1 -23903.155,E2 -23903.155} C_VEL
LIN {X 0,Y 182.777,Z 1066.278,A -85,B 0,C 180,E1 -23904.778,E2 -23904.778} C_VEL
LIN {X 0,Y 178.246,Z 1067.917,A -85,B 0,C 180,E1 -23906.497,E2 -23906.497} C_VEL
LIN {X 0,Y 174.039,Z 1069.135,A -85,B 0,C 180,E1 -23908.335,E2 -23908.335} C_VEL
LIN {X 0,Y 169.204,Z 1069.986,A -85,B 0,C 180,E1 -23910.72,E2 -23910.72} C_VEL
LIN {X 0,Y 162.897,Z 1070.025,A -85,B 0,C 180,E1 -23914.442,E2 -23914.442} C_VEL
LIN {X 0,Y 159.783,Z 1069.481,A -85,B 0,C 180,E1 -23916.681,E2 -23916.681} C_VEL
LIN {X 0,Y 154.86,Z 1067.051,A -85,B 0,C 180,E1 -23921.479,E2 -23921.479} C_VEL
LIN {X 0,Y 152.191,Z 1064.109,A -85,B 0,C 180,E1 -23925.288,E2 -23925.288} C_VEL
LIN {X 0,Y 150.174,Z 1059.963,A -85,B 0,C 180,E1 -23929.35,E2 -23929.35} C_VEL
LIN {X 0,Y 149.307,Z 1055.015,A -85,B 0,C 180,E1 -23933.243,E2 -23933.243} C_VEL
LIN {X 0,Y 149.096,Z 1048.594,A -85,B 0,C 180,E1 -23937.299,E2 -23937.299} C_VEL
LIN {X 0,Y 149.257,Z 1041.912,A -85,B 0,C 180,E1 -23940.676,E2 -23940.676} C_VEL
LIN {X 0,Y 149.581,Z 1033.402,A -85,B 0,C 180,E1 -23944.043,E2 -23944.043} C_VEL
LIN {X 0,Y 150.055,Z 1025.148,A -85,B 0,C 180,E1 -23946.725,E2 -23946.725} C_VEL
LIN {X 0,Y 150.68,Z 1015.088,A -85,B 0,C 180,E1 -23949.397,E2 -23949.397} C_VEL
LIN {X 0,Y 151.362,Z 1003.997,A -85,B 0,C 180,E1 -23951.661,E2 -23951.661} C_VEL
LIN {X 0,Y 151.976,Z 993.094,A -85,B 0,C 180,E1 -23953.37,E2 -23953.37} C_VEL
LIN {X 0,Y 152.345,Z 981.802,A -85,B 0,C 180,E1 -23954.657,E2 -23954.657} C_VEL
LIN {X 0,Y 153.531,Z 944.516,A -85,B 0,C 180,E1 -23958.086,E2 -23958.086} C_VEL
LIN {X 0,Y 153.73,Z 935.477,A -85,B 0,C 180,E1 -23958.892,E2 -23958.892} C_VEL
LIN {X 0,Y 151.579,Z 921.14,A -85,B 0,C 180,E1 -23960.082,E2 -23960.082} C_VEL
LIN {X 0,Y 150.735,Z 916.509,A -85,B 0,C 180,E1 -23960.536,E2 -23960.536} C_VEL
LIN {X 0,Y 150.213,Z 916.583,A -85,B 0,C 180,E1 -23967.898,E2 -23967.898} C_VEL
LIN {X 0,Y 150.209,Z 916.584,A -85,B 0,C 180,E1 -23972.629,E2 -23972.629} C_VEL
LIN {X 0,Y 150.17,Z 916.589,A -85,B 0,C 180,E1 -23977.476,E2 -23977.476} C_VEL
LIN {X 0,Y 150.134,Z 916.593,A -85,B 0,C 180,E1 -23981.498,E2 -23981.498} C_VEL
LIN {X 0,Y 150.128,Z 916.596,A -85,B 0,C 180,E1 -23985.397,E2 -23985.397} C_VEL
LIN {X 0,Y 150.139,Z 916.589,A -85,B 0,C 180,E1 -23989.055,E2 -23989.055} C_VEL
LIN {X 0,Y 150.178,Z 916.591,A -85,B 0,C 180,E1 -23992.711,E2 -23992.711} C_VEL
LIN {X 0,Y 150.208,Z 916.579,A -85,B 0,C 180,E1 -23997.375,E2 -23997.375} C_VEL
LIN {X 0,Y 150.242,Z 916.584,A -85,B 0,C 180,E1 -24002.724,E2 -24002.724} C_VEL
LIN {X 0,Y 150.288,Z 916.576,A -85,B 0,C 180,E1 -24009.276,E2 -24009.276} C_VEL
LIN {X 0,Y 150.324,Z 916.569,A -85,B 0,C 180,E1 -24013.71,E2 -24013.71} C_VEL
LIN {X 0,Y 150.612,Z 916.535,A -85,B 0,C 180,E1 -24019.243,E2 -24019.243} C_VEL
LIN {X 0,Y 150.701,Z 916.524,A -85,B 0,C 180,E1 -24021.958,E2 -24021.958} C_VEL
LIN {X 0,Y 151.195,Z 916.465,A -85,B 0,C 180,E1 -24030,E2 -24030} C_VEL
LIN {X 0,Y 150.701,Z 916.524,A -85,B 0,C 180,E1 -24038.043,E2 -24038.043} C_VEL
LIN {X 0,Y 150.578,Z 916.538,A -85,B 0,C 180,E1 -24041.429,E2 -24041.429} C_VEL
LIN {X 0,Y 150.315,Z 916.571,A -85,B 0,C 180,E1 -24046.292,E2 -24046.292} C_VEL
LIN {X 0,Y 150.286,Z 916.576,A -85,B 0,C 180,E1 -24050.722,E2 -24050.722} C_VEL
LIN {X 0,Y 150.189,Z 916.591,A -85,B 0,C 180,E1 -24057.237,E2 -24057.237} C_VEL
LIN {X 0,Y 150.209,Z 916.578,A -85,B 0,C 180,E1 -24062.626,E2 -24062.626} C_VEL
LIN {X 0,Y 150.173,Z 916.592,A -85,B 0,C 180,E1 -24067.474,E2 -24067.474} C_VEL
LIN {X 0,Y 150.136,Z 916.589,A -85,B 0,C 180,E1 -24071.496,E2 -24071.496} C_VEL
LIN {X 0,Y 150.13,Z 916.595,A -85,B 0,C 180,E1 -24075.395,E2 -24075.395} C_VEL
LIN {X 0,Y 150.141,Z 916.591,A -85,B 0,C 180,E1 -24079.053,E2 -24079.053} C_VEL
LIN {X 0,Y 150.179,Z 916.589,A -85,B 0,C 180,E1 -24082.709,E2 -24082.709} C_VEL
LIN {X 0,Y 150.212,Z 916.584,A -85,B 0,C 180,E1 -24087.371,E2 -24087.371} C_VEL
LIN {X 0,Y 150.188,Z 916.588,A -85,B 0,C 180,E1 -24092.762,E2 -24092.762} C_VEL
LIN {X 0,Y 150.285,Z 916.571,A -85,B 0,C 180,E1 -24099.277,E2 -24099.277} C_VEL
LIN {X 0,Y 150.317,Z 916.573,A -85,B 0,C 180,E1 -24103.707,E2 -24103.707} C_VEL
LIN {X 0,Y 150.609,Z 916.53,A -85,B 0,C 180,E1 -24109.241,E2 -24109.241} C_VEL
LIN {X 0,Y 150.699,Z 916.526,A -85,B 0,C 180,E1 -24111.956,E2 -24111.956} C_VEL
LIN {X 0,Y 151.193,Z 916.462,A -85,B 0,C 180,E1 -24119.999,E2 -24119.999} C_VEL
LIN {X 0,Y 150.681,Z 916.522,A -85,B 0,C 180,E1 -24128.042,E2 -24128.042} C_VEL
LIN {X 0,Y 150.574,Z 916.54,A -85,B 0,C 180,E1 -24131.426,E2 -24131.426} C_VEL
LIN {X 0,Y 150.315,Z 916.567,A -85,B 0,C 180,E1 -24136.291,E2 -24136.291} C_VEL
LIN {X 0,Y 150.282,Z 916.578,A -85,B 0,C 180,E1 -24140.72,E2 -24140.72} C_VEL
LIN {X 0,Y 150.185,Z 916.587,A -85,B 0,C 180,E1 -24147.236,E2 -24147.236} C_VEL
LIN {X 0,Y 150.208,Z 916.584,A -85,B 0,C 180,E1 -24152.627,E2 -24152.627} C_VEL
LIN {X 0,Y 150.168,Z 916.59,A -85,B 0,C 180,E1 -24157.473,E2 -24157.473} C_VEL
LIN {X 0,Y 150.133,Z 916.595,A -85,B 0,C 180,E1 -24161.496,E2 -24161.496} C_VEL
LIN {X 0,Y 150.125,Z 916.592,A -85,B 0,C 180,E1 -24165.394,E2 -24165.394} C_VEL
LIN {X 0,Y 150.136,Z 916.594,A -85,B 0,C 180,E1 -24169.053,E2 -24169.053} C_VEL
LIN {X 0,Y 150.174,Z 916.584,A -85,B 0,C 180,E1 -24172.709,E2 -24172.709} C_VEL
LIN {X 0,Y 150.338,Z 916.569,A -85,B 0,C 180,E1 -24179.053,E2 -24179.053} C_VEL
LIN {X 0,Y 151.301,Z 916.47,A -85,B 0,C 180,E1 -24185.653,E2 -24185.653} C_VEL
LIN {X 0,Y 150.749,Z 921.076,A -85,B 0,C 180,E1 -24188.698,E2 -24188.698} C_VEL
LIN {X 0,Y 151.131,Z 940.059,A -85,B 0,C 180,E1 -24190.395,E2 -24190.395} C_VEL
LIN {X 0,Y 153.483,Z 967.568,A -85,B 0,C 180,E1 -24192.77,E2 -24192.77} C_VEL
LIN {X 0,Y 152.765,Z 1000.267,A -85,B 0,C 180,E1 -24195.906,E2 -24195.906} C_VEL
LIN {X 0,Y 152.233,Z 1012.79,A -85,B 0,C 180,E1 -24197.671,E2 -24197.671} C_VEL
LIN {X 0,Y 151.826,Z 1021.668,A -85,B 0,C 180,E1 -24199.329,E2 -24199.329} C_VEL
LIN {X 0,Y 151.445,Z 1030.297,A -85,B 0,C 180,E1 -24201.325,E2 -24201.325} C_VEL
LIN {X 0,Y 151.122,Z 1039.574,A -85,B 0,C 180,E1 -24203.993,E2 -24203.993} C_VEL
LIN {X 0,Y 150.93,Z 1048.641,A -85,B 0,C 180,E1 -24207.331,E2 -24207.331} C_VEL
LIN {X 0,Y 150.761,Z 1054.457,A -85,B 0,C 180,E1 -24209.999,E2 -24209.999} C_VEL
LIN {X 0,Y 150.378,Z 1059.202,A -85,B 0,C 180,E1 -24212.678,E2 -24212.678} C_VEL
LIN {X 0,Y 149.773,Z 1064.587,A -85,B 0,C 180,E1 -24216.736,E2 -24216.736} C_VEL
LIN {X 0,Y 149.91,Z 1068.805,A -85,B 0,C 180,E1 -24220.808,E2 -24220.808} C_VEL
LIN {X 0,Y 150.41,Z 1071.019,A -85,B 0,C 180,E1 -24223.51,E2 -24223.51} C_VEL
LIN {X 0,Y 151.456,Z 1072.814,A -85,B 0,C 180,E1 -24226.165,E2 -24226.165} C_VEL
LIN {X 0,Y 154.89,Z 1075.14,A -85,B 0,C 180,E1 -24231.284,E2 -24231.284} C_VEL
LIN {X 0,Y 157.133,Z 1075.751,A -85,B 0,C 180,E1 -24233.737,E2 -24233.737} C_VEL
LIN {X 0,Y 162.944,Z 1075.719,A -85,B 0,C 180,E1 -24238.323,E2 -24238.323} C_VEL
LIN {X 0,Y 166.437,Z 1075.172,A -85,B 0,C 180,E1 -24240.445,E2 -24240.445} C_VEL
LIN {X 0,Y 174.392,Z 1072.711,A -85,B 0,C 180,E1 -24244.346,E2 -24244.346} C_VEL
LIN {X 0,Y 181.123,Z 1069.779,A -85,B 0,C 180,E1 -24246.973,E2 -24246.973} C_VEL
LIN {X 0,Y 188.43,Z 1065.775,A -85,B 0,C 180,E1 -24249.35,E2 -24249.35} C_VEL
LIN {X 0,Y 196.235,Z 1060.64,A -85,B 0,C 180,E1 -24251.495,E2 -24251.495} C_VEL
LIN {X 0,Y 200.049,Z 1057.809,A -85,B 0,C 180,E1 -24252.379,E2 -24252.379} C_VEL
LIN {X 0,Y 201.098,Z 1056.861,A -85,B 0,C 180,E1 -24252.906,E2 -24252.906} C_VEL
LIN {X 0,Y 201.277,Z 1056.449,A -85,B 0,C 180,E1 -24253.835,E2 -24253.835} C_VEL
LIN {X 0,Y 200.173,Z 1056.91,A -85,B 0,C 180,E1 -24255.11,E2 -24255.11} C_VEL
LIN {X 0,Y 198.602,Z 1057.774,A -85,B 0,C 180,E1 -24256.069,E2 -24256.069} C_VEL
LIN {X 0,Y 196.124,Z 1059.218,A -85,B 0,C 180,E1 -24257.195,E2 -24257.195} C_VEL
LIN {X 0,Y 191.975,Z 1061.623,A -85,B 0,C 180,E1 -24258.797,E2 -24258.797} C_VEL
LIN {X 0,Y 187.29,Z 1063.977,A -85,B 0,C 180,E1 -24260.278,E2 -24260.278} C_VEL
LIN {X 0,Y 182.048,Z 1066.261,A -85,B 0,C 180,E1 -24261.854,E2 -24261.854} C_VEL
LIN {X 0,Y 177.155,Z 1068.035,A -85,B 0,C 180,E1 -24263.483,E2 -24263.483} C_VEL
LIN {X 0,Y 172.46,Z 1069.351,A -85,B 0,C 180,E1 -24265.215,E2 -24265.215} C_VEL
LIN {X 0,Y 163.952,Z 1070.561,A -85,B 0,C 180,E1 -24269.044,E2 -24269.044} C_VEL
LIN {X 0,Y 160.082,Z 1070.613,A -85,B 0,C 180,E1 -24271.124,E2 -24271.124} C_VEL
LIN {X 0,Y 153.316,Z 1069.269,A -85,B 0,C 180,E1 -24275.636,E2 -24275.636} C_VEL
LIN {X 0,Y 150.542,Z 1068.07,A -85,B 0,C 180,E1 -24278.071,E2 -24278.071} C_VEL
LIN {X 0,Y 147.198,Z 1065.385,A -85,B 0,C 180,E1 -24281.921,E2 -24281.921} C_VEL
LIN {X 0,Y 144.68,Z 1061.711,A -85,B 0,C 180,E1 -24285.945,E2 -24285.945} C_VEL
LIN {X 0,Y 142.981,Z 1056.881,A -85,B 0,C 180,E1 -24290.095,E2 -24290.095} C_VEL
LIN {X 0,Y 142.369,Z 1050.956,A -85,B 0,C 180,E1 -24294.335,E2 -24294.335} C_VEL
LIN {X 0,Y 142.371,Z 1044.787,A -85,B 0,C 180,E1 -24297.88,E2 -24297.88} C_VEL
LIN {X 0,Y 142.57,Z 1037.269,A -85,B 0,C 180,E1 -24301.414,E2 -24301.414} C_VEL
LIN {X 0,Y 143.005,Z 1027.858,A -85,B 0,C 180,E1 -24304.935,E2 -24304.935} C_VEL
LIN {X 0,Y 143.558,Z 1018.314,A -85,B 0,C 180,E1 -24307.738,E2 -24307.738} C_VEL
LIN {X 0,Y 144.179,Z 1007.987,A -85,B 0,C 180,E1 -24310.179,E2 -24310.179} C_VEL
LIN {X 0,Y 144.873,Z 996.367,A -85,B 0,C 180,E1 -24312.266,E2 -24312.266} C_VEL
LIN {X 0,Y 145.406,Z 984.908,A -85,B 0,C 180,E1 -24313.788,E2 -24313.788} C_VEL
LIN {X 0,Y 146.566,Z 941.754,A -85,B 0,C 180,E1 -24318.072,E2 -24318.072} C_VEL
LIN {X 0,Y 146.583,Z 934.922,A -85,B 0,C 180,E1 -24318.7,E2 -24318.7} C_VEL
LIN {X 0,Y 144.61,Z 922.262,A -85,B 0,C 180,E1 -24319.805,E2 -24319.805} C_VEL
LIN {X 0,Y 143.745,Z 917.381,A -85,B 0,C 180,E1 -24320.245,E2 -24320.245} C_VEL
LIN {X 0,Y 143.184,Z 917.458,A -85,B 0,C 180,E1 -24327.932,E2 -24327.932} C_VEL
LIN {X 0,Y 143.139,Z 917.467,A -85,B 0,C 180,E1 -24333.418,E2 -24333.418} C_VEL
LIN {X 0,Y 143.053,Z 917.472,A -85,B 0,C 180,E1 -24339.695,E2 -24339.695} C_VEL
LIN {X 0,Y 143.035,Z 917.48,A -85,B 0,C 180,E1 -24343.465,E2 -24343.465} C_VEL
LIN {X 0,Y 143.039,Z 917.475,A -85,B 0,C 180,E1 -24347.479,E2 -24347.479} C_VEL
LIN {X 0,Y 143.074,Z 917.474,A -85,B 0,C 180,E1 -24351.811,E2 -24351.811} C_VEL
LIN {X 0,Y 143.175,Z 917.455,A -85,B 0,C 180,E1 -24357.32,E2 -24357.32} C_VEL
LIN {X 0,Y 143.185,Z 917.461,A -85,B 0,C 180,E1 -24362.07,E2 -24362.07} C_VEL
LIN {X 0,Y 143.226,Z 917.453,A -85,B 0,C 180,E1 -24368.803,E2 -24368.803} C_VEL
LIN {X 0,Y 143.262,Z 917.452,A -85,B 0,C 180,E1 -24372.882,E2 -24372.882} C_VEL
LIN {X 0,Y 143.538,Z 917.415,A -85,B 0,C 180,E1 -24378.706,E2 -24378.706} C_VEL
LIN {X 0,Y 143.624,Z 917.408,A -85,B 0,C 180,E1 -24381.559,E2 -24381.559} C_VEL
LIN {X 0,Y 144.153,Z 917.342,A -85,B 0,C 180,E1 -24390.001,E2 -24390.001} C_VEL
LIN {X 0,Y 143.623,Z 917.408,A -85,B 0,C 180,E1 -24398.442,E2 -24398.442} C_VEL
LIN {X 0,Y 143.502,Z 917.419,A -85,B 0,C 180,E1 -24401.615,E2 -24401.615} C_VEL
LIN {X 0,Y 143.256,Z 917.453,A -85,B 0,C 180,E1 -24407.119,E2 -24407.119} C_VEL
LIN {X 0,Y 143.222,Z 917.453,A -85,B 0,C 180,E1 -24411.193,E2 -24411.193} C_VEL
LIN {X 0,Y 143.146,Z 917.466,A -85,B 0,C 180,E1 -24417.9,E2 -24417.9} C_VEL
LIN {X 0,Y 143.14,Z 917.461,A -85,B 0,C 180,E1 -24423.415,E2 -24423.415} C_VEL
LIN {X 0,Y 143.056,Z 917.474,A -85,B 0,C 180,E1 -24429.693,E2 -24429.693} C_VEL
LIN {X 0,Y 143.037,Z 917.476,A -85,B 0,C 180,E1 -24433.463,E2 -24433.463} C_VEL
LIN {X 0,Y 143.041,Z 917.479,A -85,B 0,C 180,E1 -24437.477,E2 -24437.477} C_VEL
LIN {X 0,Y 143.075,Z 917.469,A -85,B 0,C 180,E1 -24441.809,E2 -24441.809} C_VEL
LIN {X 0,Y 143.179,Z 917.46,A -85,B 0,C 180,E1 -24447.319,E2 -24447.319} C_VEL
LIN {X 0,Y 143.109,Z 917.47,A -85,B 0,C 180,E1 -24453.768,E2 -24453.768} C_VEL
LIN {X 0,Y 143.249,Z 917.448,A -85,B 0,C 180,E1 -24459.912,E2 -24459.912} C_VEL
LIN {X 0,Y 143.309,Z 917.444,A -85,B 0,C 180,E1 -24465.805,E2 -24465.805} C_VEL
LIN {X 0,Y 143.535,Z 917.409,A -85,B 0,C 180,E1 -24468.704,E2 -24468.704} C_VEL
LIN {X 0,Y 143.621,Z 917.406,A -85,B 0,C 180,E1 -24471.557,E2 -24471.557} C_VEL
LIN {X 0,Y 144.151,Z 917.339,A -85,B 0,C 180,E1 -24479.999,E2 -24479.999} C_VEL
LIN {X 0,Y 143.607,Z 917.405,A -85,B 0,C 180,E1 -24488.441,E2 -24488.441} C_VEL
LIN {X 0,Y 143.499,Z 917.421,A -85,B 0,C 180,E1 -24491.613,E2 -24491.613} C_VEL
LIN {X 0,Y 143.255,Z 917.448,A -85,B 0,C 180,E1 -24497.118,E2 -24497.118} C_VEL
LIN {X 0,Y 143.219,Z 917.457,A -85,B 0,C 180,E1 -24501.192,E2 -24501.192} C_VEL
LIN {X 0,Y 143.142,Z 917.465,A -85,B 0,C 180,E1 -24507.899,E2 -24507.899} C_VEL
LIN {X 0,Y 143.138,Z 917.462,A -85,B 0,C 180,E1 -24513.415,E2 -24513.415} C_VEL
LIN {X 0,Y 143.051,Z 917.48,A -85,B 0,C 180,E1 -24519.692,E2 -24519.692} C_VEL
LIN {X 0,Y 143.032,Z 917.475,A -85,B 0,C 180,E1 -24523.463,E2 -24523.463} C_VEL
LIN {X 0,Y 143.037,Z 917.479,A -85,B 0,C 180,E1 -24527.476,E2 -24527.476} C_VEL
LIN {X 0,Y 143.071,Z 917.473,A -85,B 0,C 180,E1 -24531.808,E2 -24531.808} C_VEL
LIN {X 0,Y 143.222,Z 917.456,A -85,B 0,C 180,E1 -24537.331,E2 -24537.331} C_VEL
LIN {X 0,Y 144.229,Z 917.335,A -85,B 0,C 180,E1 -24545.531,E2 -24545.531} C_VEL
LIN {X 0,Y 144.144,Z 917.475,A -85,B 0,C 180,E1 -24546.567,E2 -24546.567} C_VEL
LIN {X 0,Y 143.677,Z 920.599,A -85,B 0,C 180,E1 -24548.843,E2 -24548.843} C_VEL
LIN {X 0,Y 144.067,Z 940.045,A -85,B 0,C 180,E1 -24550.682,E2 -24550.682} C_VEL
LIN {X 0,Y 146.466,Z 967.534,A -85,B 0,C 180,E1 -24553.177,E2 -24553.177} C_VEL
LIN {X 0,Y 145.847,Z 999.419,A -85,B 0,C 180,E1 -24556.413,E2 -24556.413} C_VEL
LIN {X 0,Y 145.365,Z 1011.25,A -85,B 0,C 180,E1 -24558.142,E2 -24558.142} C_VEL
LIN {X 0,Y 144.985,Z 1021.776,A -85,B 0,C 180,E1 -24560.231,E2 -24560.231} C_VEL
LIN {X 0,Y 144.683,Z 1030.226,A -85,B 0,C 180,E1 -24562.323,E2 -24562.323} C_VEL
LIN {X 0,Y 144.404,Z 1039.404,A -85,B 0,C 180,E1 -24565.114,E2 -24565.114} C_VEL
LIN {X 0,Y 144.249,Z 1048.352,A -85,B 0,C 180,E1 -24568.604,E2 -24568.604} C_VEL
LIN {X 0,Y 144.007,Z 1053.95,A -85,B 0,C 180,E1 -24571.398,E2 -24571.398} C_VEL
LIN {X 0,Y 143.578,Z 1058.511,A -85,B 0,C 180,E1 -24574.21,E2 -24574.21} C_VEL
LIN {X 0,Y 143.058,Z 1063.869,A -85,B 0,C 180,E1 -24578.475,E2 -24578.475} C_VEL
LIN {X 0,Y 143.437,Z 1067.996,A -85,B 0,C 180,E1 -24582.737,E2 -24582.737} C_VEL
LIN {X 0,Y 144.828,Z 1071.184,A -85,B 0,C 180,E1 -24586.927,E2 -24586.927} C_VEL
LIN {X 0,Y 146.376,Z 1072.845,A -85,B 0,C 180,E1 -24589.639,E2 -24589.639} C_VEL
LIN {X 0,Y 150.726,Z 1074.839,A -85,B 0,C 180,E1 -24594.812,E2 -24594.812} C_VEL
LIN {X 0,Y 153.519,Z 1075.359,A -85,B 0,C 180,E1 -24597.244,E2 -24597.244} C_VEL
LIN {X 0,Y 156.751,Z 1075.406,A -85,B 0,C 180,E1 -24599.55,E2 -24599.55} C_VEL
LIN {X 0,Y 164.31,Z 1074.466,A -85,B 0,C 180,E1 -24603.782,E2 -24603.782} C_VEL
LIN {X 0,Y 168.59,Z 1073.339,A -85,B 0,C 180,E1 -24605.705,E2 -24605.705} C_VEL
LIN {X 0,Y 178.003,Z 1069.932,A -85,B 0,C 180,E1 -24609.177,E2 -24609.177} C_VEL
LIN {X 0,Y 185.713,Z 1066.152,A -85,B 0,C 180,E1 -24611.472,E2 -24611.472} C_VEL
LIN {X 0,Y 193.905,Z 1061.253,A -85,B 0,C 180,E1 -24613.523,E2 -24613.523} C_VEL
LIN {X 0,Y 201.203,Z 1056.111,A -85,B 0,C 180,E1 -24615.018,E2 -24615.018} C_VEL
LIN {X 0,Y 205.732,Z 1052.569,A -85,B 0,C 180,E1 -24615.838,E2 -24615.838} C_VEL
LIN {X 0,Y 197.927,Z 1058.096,A -85,B 0,C 180,E1 -24617.574,E2 -24617.574} C_VEL
LIN {X 0,Y 189.739,Z 1062.755,A -85,B 0,C 180,E1 -24619.595,E2 -24619.595} C_VEL
LIN {X 0,Y 187.29,Z 1063.977,A -85,B 0,C 180,E1 -24620.278,E2 -24620.278} C_VEL
LIN {X 0,Y 182.818,Z 1065.99,A -85,B 0,C 180,E1 -24621.315,E2 -24621.315} C_VEL
LIN {X 0,Y 174.398,Z 1068.815,A -85,B 0,C 180,E1 -24622.749,E2 -24622.749} C_VEL
LIN {X 0,Y 167.681,Z 1070.377,A -85,B 0,C 180,E1 -24624.033,E2 -24624.033} C_VEL
LIN {X 0,Y 163.199,Z 1070.973,A -85,B 0,C 180,E1 -24625.322,E2 -24625.322} C_VEL
LIN {X 0,Y 161.92,Z 1071.032,A -85,B 0,C 180,E1 -24625.841,E2 -24625.841} C_VEL
LIN {X 0,Y 157.932,Z 1071.096,A -85,B 0,C 180,E1 -24627.725,E2 -24627.725} C_VEL
LIN {X 0,Y 150.233,Z 1070.067,A -85,B 0,C 180,E1 -24632.109,E2 -24632.109} C_VEL
LIN {X 0,Y 146.897,Z 1068.924,A -85,B 0,C 180,E1 -24634.496,E2 -24634.496} C_VEL
LIN {X 0,Y 141.58,Z 1065.424,A -85,B 0,C 180,E1 -24639.668,E2 -24639.668} C_VEL
LIN {X 0,Y 138.733,Z 1061.664,A -85,B 0,C 180,E1 -24643.823,E2 -24643.823} C_VEL
LIN {X 0,Y 136.666,Z 1056.858,A -85,B 0,C 180,E1 -24648.131,E2 -24648.131} C_VEL
LIN {X 0,Y 135.696,Z 1049.771,A -85,B 0,C 180,E1 -24653.309,E2 -24653.309} C_VEL
LIN {X 0,Y 135.679,Z 1042.08,A -85,B 0,C 180,E1 -24657.775,E2 -24657.775} C_VEL
LIN {X 0,Y 135.855,Z 1035.659,A -85,B 0,C 180,E1 -24660.742,E2 -24660.742} C_VEL
LIN {X 0,Y 136.244,Z 1026.902,A -85,B 0,C 180,E1 -24664.069,E2 -24664.069} C_VEL
LIN {X 0,Y 136.66,Z 1018.648,A -85,B 0,C 180,E1 -24666.646,E2 -24666.646} C_VEL
LIN {X 0,Y 137.217,Z 1008.597,A -85,B 0,C 180,E1 -24669.212,E2 -24669.212} C_VEL
LIN {X 0,Y 137.954,Z 996.194,A -85,B 0,C 180,E1 -24671.573,E2 -24671.573} C_VEL
LIN {X 0,Y 138.467,Z 984.163,A -85,B 0,C 180,E1 -24673.235,E2 -24673.235} C_VEL
LIN {X 0,Y 139.668,Z 937.293,A -85,B 0,C 180,E1 -24678.142,E2 -24678.142} C_VEL
LIN {X 0,Y 137.769,Z 923.815,A -85,B 0,C 180,E1 -24679.388,E2 -24679.388} C_VEL
LIN {X 0,Y 136.757,Z 918.254,A -85,B 0,C 180,E1 -24679.928,E2 -24679.928} C_VEL
LIN {X 0,Y 136.093,Z 918.341,A -85,B 0,C 180,E1 -24688.611,E2 -24688.611} C_VEL
LIN {X 0,Y 136.041,Z 918.351,A -85,B 0,C 180,E1 -24694.631,E2 -24694.631} C_VEL
LIN {X 0,Y 136.025,Z 918.346,A -85,B 0,C 180,E1 -24699.195,E2 -24699.195} C_VEL
LIN {X 0,Y 135.98,Z 918.359,A -85,B 0,C 180,E1 -24703.65,E2 -24703.65} C_VEL
LIN {X 0,Y 135.984,Z 918.353,A -85,B 0,C 180,E1 -24707.789,E2 -24707.789} C_VEL
LIN {X 0,Y 136.023,Z 918.352,A -85,B 0,C 180,E1 -24711.683,E2 -24711.683} C_VEL
LIN {X 0,Y 136.054,Z 918.347,A -85,B 0,C 180,E1 -24715.743,E2 -24715.743} C_VEL
LIN {X 0,Y 136.142,Z 918.339,A -85,B 0,C 180,E1 -24722.316,E2 -24722.316} C_VEL
LIN {X 0,Y 136.189,Z 918.329,A -85,B 0,C 180,E1 -24728.825,E2 -24728.825} C_VEL
LIN {X 0,Y 136.233,Z 918.323,A -85,B 0,C 180,E1 -24735.053,E2 -24735.053} C_VEL
LIN {X 0,Y 136.429,Z 918.3,A -85,B 0,C 180,E1 -24738.178,E2 -24738.178} C_VEL
LIN {X 0,Y 136.55,Z 918.288,A -85,B 0,C 180,E1 -24741.118,E2 -24741.118} C_VEL
LIN {X 0,Y 137.11,Z 918.22,A -85,B 0,C 180,E1 -24750.001,E2 -24750.001} C_VEL
LIN {X 0,Y 136.55,Z 918.288,A -85,B 0,C 180,E1 -24758.883,E2 -24758.883} C_VEL
LIN {X 0,Y 136.418,Z 918.302,A -85,B 0,C 180,E1 -24761.893,E2 -24761.893} C_VEL
LIN {X 0,Y 136.168,Z 918.335,A -85,B 0,C 180,E1 -24768.04,E2 -24768.04} C_VEL
LIN {X 0,Y 136.147,Z 918.333,A -85,B 0,C 180,E1 -24771.689,E2 -24771.689} C_VEL
LIN {X 0,Y 136.065,Z 918.348,A -85,B 0,C 180,E1 -24778.585,E2 -24778.585} C_VEL
LIN {X 0,Y 136.043,Z 918.348,A -85,B 0,C 180,E1 -24784.63,E2 -24784.63} C_VEL
LIN {X 0,Y 136.028,Z 918.352,A -85,B 0,C 180,E1 -24789.194,E2 -24789.194} C_VEL
LIN {X 0,Y 135.982,Z 918.355,A -85,B 0,C 180,E1 -24793.648,E2 -24793.648} C_VEL
LIN {X 0,Y 135.986,Z 918.358,A -85,B 0,C 180,E1 -24797.787,E2 -24797.787} C_VEL
LIN {X 0,Y 136.024,Z 918.347,A -85,B 0,C 180,E1 -24801.681,E2 -24801.681} C_VEL
LIN {X 0,Y 136.056,Z 918.349,A -85,B 0,C 180,E1 -24805.741,E2 -24805.741} C_VEL
LIN {X 0,Y 136.065,Z 918.345,A -85,B 0,C 180,E1 -24811.413,E2 -24811.413} C_VEL
LIN {X 0,Y 136.184,Z 918.327,A -85,B 0,C 180,E1 -24818.822,E2 -24818.822} C_VEL
LIN {X 0,Y 136.227,Z 918.329,A -85,B 0,C 180,E1 -24825.05,E2 -24825.05} C_VEL
LIN {X 0,Y 136.428,Z 918.294,A -85,B 0,C 180,E1 -24828.177,E2 -24828.177} C_VEL
LIN {X 0,Y 136.548,Z 918.286,A -85,B 0,C 180,E1 -24831.116,E2 -24831.116} C_VEL
LIN {X 0,Y 137.108,Z 918.216,A -85,B 0,C 180,E1 -24839.999,E2 -24839.999} C_VEL
LIN {X 0,Y 136.536,Z 918.288,A -85,B 0,C 180,E1 -24848.882,E2 -24848.882} C_VEL
LIN {X 0,Y 136.415,Z 918.304,A -85,B 0,C 180,E1 -24851.891,E2 -24851.891} C_VEL
LIN {X 0,Y 136.166,Z 918.332,A -85,B 0,C 180,E1 -24858.039,E2 -24858.039} C_VEL
LIN {X 0,Y 136.143,Z 918.337,A -85,B 0,C 180,E1 -24861.688,E2 -24861.688} C_VEL
LIN {X 0,Y 136.062,Z 918.347,A -85,B 0,C 180,E1 -24868.585,E2 -24868.585} C_VEL
LIN {X 0,Y 136.04,Z 918.343,A -85,B 0,C 180,E1 -24874.628,E2 -24874.628} C_VEL
LIN {X 0,Y 136.024,Z 918.353,A -85,B 0,C 180,E1 -24879.193,E2 -24879.193} C_VEL
LIN {X 0,Y 135.977,Z 918.353,A -85,B 0,C 180,E1 -24883.647,E2 -24883.647} C_VEL
LIN {X 0,Y 135.981,Z 918.359,A -85,B 0,C 180,E1 -24887.786,E2 -24887.786} C_VEL
LIN {X 0,Y 136.02,Z 918.351,A -85,B 0,C 180,E1 -24891.681,E2 -24891.681} C_VEL
LIN {X 0,Y 136.088,Z 918.343,A -85,B 0,C 180,E1 -24895.717,E2 -24895.717} C_VEL
LIN {X 0,Y 136.58,Z 918.277,A -85,B 0,C 180,E1 -24902.411,E2 -24902.411} C_VEL
LIN {X 0,Y 137.167,Z 918.214,A -85,B 0,C 180,E1 -24905.801,E2 -24905.801} C_VEL
LIN {X 0,Y 136.783,Z 918.473,A -85,B 0,C 180,E1 -24907.643,E2 -24907.643} C_VEL
LIN {X 0,Y 136.622,Z 920.436,A -85,B 0,C 180,E1 -24909.091,E2 -24909.091} C_VEL
LIN {X 0,Y 136.984,Z 939.13,A -85,B 0,C 180,E1 -24910.957,E2 -24910.957} C_VEL
LIN {X 0,Y 139.5,Z 967.885,A -85,B 0,C 180,E1 -24913.72,E2 -24913.72} C_VEL
LIN {X 0,Y 138.971,Z 999.118,A -85,B 0,C 180,E1 -24917.124,E2 -24917.124} C_VEL
LIN {X 0,Y 138.529,Z 1011.378,A -85,B 0,C 180,E1 -24919.032,E2 -24919.032} C_VEL
LIN {X 0,Y 138.189,Z 1021.77,A -85,B 0,C 180,E1 -24921.223,E2 -24921.223} C_VEL
LIN {X 0,Y 137.836,Z 1032.648,A -85,B 0,C 180,E1 -24924.146,E2 -24924.146} C_VEL
LIN {X 0,Y 137.697,Z 1040.99,A -85,B 0,C 180,E1 -24927.074,E2 -24927.074} C_VEL
LIN {X 0,Y 137.647,Z 1047.796,A -85,B 0,C 180,E1 -24929.999,E2 -24929.999} C_VEL
LIN {X 0,Y 137.332,Z 1053.285,A -85,B 0,C 180,E1 -24932.933,E2 -24932.933} C_VEL
LIN {X 0,Y 136.783,Z 1057.753,A -85,B 0,C 180,E1 -24935.898,E2 -24935.898} C_VEL
LIN {X 0,Y 136.526,Z 1063.073,A -85,B 0,C 180,E1 -24940.47,E2 -24940.47} C_VEL
LIN {X 0,Y 137.174,Z 1067.163,A -85,B 0,C 180,E1 -24944.843,E2 -24944.843} C_VEL
LIN {X 0,Y 138.261,Z 1069.434,A -85,B 0,C 180,E1 -24947.757,E2 -24947.757} C_VEL
LIN {X 0,Y 141.977,Z 1072.724,A -85,B 0,C 180,E1 -24953.328,E2 -24953.328} C_VEL
LIN {X 0,Y 144.375,Z 1073.835,A -85,B 0,C 180,E1 -24955.983,E2 -24955.983} C_VEL
LIN {X 0,Y 150.638,Z 1074.883,A -85,B 0,C 180,E1 -24960.877,E2 -24960.877} C_VEL
LIN {X 0,Y 154.401,Z 1074.916,A -85,B 0,C 180,E1 -24963.107,E2 -24963.107} C_VEL
LIN {X 0,Y 162.878,Z 1073.727,A -85,B 0,C 180,E1 -24967.163,E2 -24967.163} C_VEL
LIN {X 0,Y 167.623,Z 1072.598,A -85,B 0,C 180,E1 -24968.969,E2 -24968.969} C_VEL
LIN {X 0,Y 177.806,Z 1068.977,A -85,B 0,C 180,E1 -24972.217,E2 -24972.217} C_VEL
LIN {X 0,Y 186.324,Z 1064.989,A -85,B 0,C 180,E1 -24974.402,E2 -24974.402} C_VEL
LIN {X 0,Y 190.634,Z 1062.68,A -85,B 0,C 180,E1 -24975.352,E2 -24975.352} C_VEL
LIN {X 0,Y 192.985,Z 1061.179,A -85,B 0,C 180,E1 -24976.218,E2 -24976.218} C_VEL
LIN {X 0,Y 183.192,Z 1065.821,A -85,B 0,C 180,E1 -24978.584,E2 -24978.584} C_VEL
LIN {X 0,Y 176.664,Z 1068.197,A -85,B 0,C 180,E1 -24980.469,E2 -24980.469} C_VEL
LIN {X 0,Y 171.572,Z 1069.536,A -85,B 0,C 180,E1 -24982.09,E2 -24982.09} C_VEL
LIN {X 0,Y 162.196,Z 1071.027,A -85,B 0,C 180,E1 -24985.717,E2 -24985.717} C_VEL
LIN {X 0,Y 161.92,Z 1071.032,A -85,B 0,C 180,E1 -24985.841,E2 -24985.841} C_VEL
LIN {X 0,Y 157.83,Z 1071.161,A -85,B 0,C 180,E1 -24987.372,E2 -24987.372} C_VEL
LIN {X 0,Y 150.04,Z 1070.663,A -85,B 0,C 180,E1 -24989.653,E2 -24989.653} C_VEL
LIN {X 0,Y 144.067,Z 1069.466,A -85,B 0,C 180,E1 -24991.629,E2 -24991.629} C_VEL
LIN {X 0,Y 140.457,Z 1068.186,A -85,B 0,C 180,E1 -24993.432,E2 -24993.432} C_VEL
LIN {X 0,Y 139.539,Z 1067.685,A -85,B 0,C 180,E1 -24994.116,E2 -24994.116} C_VEL
LIN {X 0,Y 136.275,Z 1065.372,A -85,B 0,C 180,E1 -24997.246,E2 -24997.246} C_VEL
LIN {X 0,Y 133.039,Z 1061.592,A -85,B 0,C 180,E1 -25001.522,E2 -25001.522} C_VEL
LIN {X 0,Y 130.674,Z 1056.865,A -85,B 0,C 180,E1 -25005.833,E2 -25005.833} C_VEL
LIN {X 0,Y 129.312,Z 1050.733,A -85,B 0,C 180,E1 -25010.618,E2 -25010.618} C_VEL
LIN {X 0,Y 129.059,Z 1043.351,A -85,B 0,C 180,E1 -25015.316,E2 -25015.316} C_VEL
LIN {X 0,Y 129.219,Z 1035.632,A -85,B 0,C 180,E1 -25019.222,E2 -25019.222} C_VEL
LIN {X 0,Y 129.396,Z 1028.072,A -85,B 0,C 180,E1 -25022.336,E2 -25022.336} C_VEL
LIN {X 0,Y 129.807,Z 1020.08,A -85,B 0,C 180,E1 -25025.049,E2 -25025.049} C_VEL
LIN {X 0,Y 130.326,Z 1010.333,A -85,B 0,C 180,E1 -25027.749,E2 -25027.749} C_VEL
LIN {X 0,Y 130.976,Z 997.737,A -85,B 0,C 180,E1 -25030.435,E2 -25030.435} C_VEL
LIN {X 0,Y 131.501,Z 986.767,A -85,B 0,C 180,E1 -25032.15,E2 -25032.15} C_VEL
LIN {X 0,Y 132.383,Z 946.008,A -85,B 0,C 180,E1 -25036.779,E2 -25036.779} C_VEL
LIN {X 0,Y 132.584,Z 935.992,A -85,B 0,C 180,E1 -25037.856,E2 -25037.856} C_VEL
LIN {X 0,Y 130.516,Z 923.477,A -85,B 0,C 180,E1 -25039.055,E2 -25039.055} C_VEL
LIN {X 0,Y 129.77,Z 919.126,A -85,B 0,C 180,E1 -25039.58,E2 -25039.58} C_VEL
LIN {X 0,Y 129.076,Z 919.218,A -85,B 0,C 180,E1 -25045.824,E2 -25045.824} C_VEL
LIN {X 0,Y 129.018,Z 919.219,A -85,B 0,C 180,E1 -25049.359,E2 -25049.359} C_VEL
LIN {X 0,Y 128.957,Z 919.234,A -85,B 0,C 180,E1 -25055.167,E2 -25055.167} C_VEL
LIN {X 0,Y 128.924,Z 919.234,A -85,B 0,C 180,E1 -25060.858,E2 -25060.858} C_VEL
LIN {X 0,Y 128.913,Z 919.238,A -85,B 0,C 180,E1 -25065.133,E2 -25065.133} C_VEL
LIN {X 0,Y 128.936,Z 919.23,A -85,B 0,C 180,E1 -25069.742,E2 -25069.742} C_VEL
LIN {X 0,Y 128.958,Z 919.232,A -85,B 0,C 180,E1 -25074.836,E2 -25074.836} C_VEL
LIN {X 0,Y 129.02,Z 919.225,A -85,B 0,C 180,E1 -25080.643,E2 -25080.643} C_VEL
LIN {X 0,Y 129.012,Z 919.226,A -85,B 0,C 180,E1 -25084.164,E2 -25084.164} C_VEL
LIN {X 0,Y 129.072,Z 919.214,A -85,B 0,C 180,E1 -25087.771,E2 -25087.771} C_VEL
LIN {X 0,Y 129.154,Z 919.206,A -85,B 0,C 180,E1 -25094.213,E2 -25094.213} C_VEL
LIN {X 0,Y 129.348,Z 919.183,A -85,B 0,C 180,E1 -25097.97,E2 -25097.97} C_VEL
LIN {X 0,Y 129.473,Z 919.169,A -85,B 0,C 180,E1 -25100.629,E2 -25100.629} C_VEL
LIN {X 0,Y 130.065,Z 919.097,A -85,B 0,C 180,E1 -25110.001,E2 -25110.001} C_VEL
LIN {X 0,Y 129.473,Z 919.169,A -85,B 0,C 180,E1 -25119.373,E2 -25119.373} C_VEL
LIN {X 0,Y 129.301,Z 919.185,A -85,B 0,C 180,E1 -25122.558,E2 -25122.558} C_VEL
LIN {X 0,Y 129.085,Z 919.218,A -85,B 0,C 180,E1 -25129.067,E2 -25129.067} C_VEL
LIN {X 0,Y 129.037,Z 919.218,A -85,B 0,C 180,E1 -25132.412,E2 -25132.412} C_VEL
LIN {X 0,Y 129.003,Z 919.227,A -85,B 0,C 180,E1 -25139.362,E2 -25139.362} C_VEL
LIN {X 0,Y 128.959,Z 919.232,A -85,B 0,C 180,E1 -25145.165,E2 -25145.165} C_VEL
LIN {X 0,Y 128.926,Z 919.231,A -85,B 0,C 180,E1 -25150.856,E2 -25150.856} C_VEL
LIN {X 0,Y 128.915,Z 919.238,A -85,B 0,C 180,E1 -25155.131,E2 -25155.131} C_VEL
LIN {X 0,Y 128.937,Z 919.231,A -85,B 0,C 180,E1 -25159.739,E2 -25159.739} C_VEL
LIN {X 0,Y 128.96,Z 919.234,A -85,B 0,C 180,E1 -25164.833,E2 -25164.833} C_VEL
LIN {X 0,Y 129.003,Z 919.221,A -85,B 0,C 180,E1 -25170.655,E2 -25170.655} C_VEL
LIN {X 0,Y 129.07,Z 919.215,A -85,B 0,C 180,E1 -25177.772,E2 -25177.772} C_VEL
LIN {X 0,Y 129.149,Z 919.209,A -85,B 0,C 180,E1 -25184.21,E2 -25184.21} C_VEL
LIN {X 0,Y 129.346,Z 919.177,A -85,B 0,C 180,E1 -25187.971,E2 -25187.971} C_VEL
LIN {X 0,Y 129.471,Z 919.167,A -85,B 0,C 180,E1 -25190.626,E2 -25190.626} C_VEL
LIN {X 0,Y 130.063,Z 919.094,A -85,B 0,C 180,E1 -25199.999,E2 -25199.999} C_VEL
LIN {X 0,Y 129.462,Z 919.168,A -85,B 0,C 180,E1 -25209.371,E2 -25209.371} C_VEL
LIN {X 0,Y 129.298,Z 919.192,A -85,B 0,C 180,E1 -25212.556,E2 -25212.556} C_VEL
LIN {X 0,Y 129.082,Z 919.218,A -85,B 0,C 180,E1 -25219.066,E2 -25219.066} C_VEL
LIN {X 0,Y 129.034,Z 919.223,A -85,B 0,C 180,E1 -25222.411,E2 -25222.411} C_VEL
LIN {X 0,Y 128.999,Z 919.23,A -85,B 0,C 180,E1 -25229.361,E2 -25229.361} C_VEL
LIN {X 0,Y 128.956,Z 919.226,A -85,B 0,C 180,E1 -25235.164,E2 -25235.164} C_VEL
LIN {X 0,Y 128.922,Z 919.237,A -85,B 0,C 180,E1 -25240.855,E2 -25240.855} C_VEL
LIN {X 0,Y 128.911,Z 919.234,A -85,B 0,C 180,E1 -25245.131,E2 -25245.131} C_VEL
LIN {X 0,Y 128.933,Z 919.237,A -85,B 0,C 180,E1 -25249.739,E2 -25249.739} C_VEL
LIN {X 0,Y 129.069,Z 919.22,A -85,B 0,C 180,E1 -25257.008,E2 -25257.008} C_VEL
LIN {X 0,Y 129.812,Z 919.129,A -85,B 0,C 180,E1 -25264.334,E2 -25264.334} C_VEL
LIN {X 0,Y 129.67,Z 919.146,A -85,B 0,C 180,E1 -25267.703,E2 -25267.703} C_VEL
LIN {X 0,Y 129.561,Z 919.246,A -85,B 0,C 180,E1 -25268.729,E2 -25268.729} C_VEL
LIN {X 0,Y 129.564,Z 920.012,A -85,B 0,C 180,E1 -25269.354,E2 -25269.354} C_VEL
LIN {X 0,Y 129.995,Z 939.15,A -85,B 0,C 180,E1 -25271.427,E2 -25271.427} C_VEL
LIN {X 0,Y 132.544,Z 967.859,A -85,B 0,C 180,E1 -25274.339,E2 -25274.339} C_VEL
LIN {X 0,Y 132.106,Z 998.778,A -85,B 0,C 180,E1 -25277.908,E2 -25277.908} C_VEL
LIN {X 0,Y 131.746,Z 1011.421,A -85,B 0,C 180,E1 -25280.015,E2 -25280.015} C_VEL
LIN {X 0,Y 131.496,Z 1021.549,A -85,B 0,C 180,E1 -25282.321,E2 -25282.321} C_VEL
LIN {X 0,Y 131.203,Z 1032.134,A -85,B 0,C 180,E1 -25285.391,E2 -25285.391} C_VEL
LIN {X 0,Y 131.165,Z 1040.467,A -85,B 0,C 180,E1 -25288.464,E2 -25288.464} C_VEL
LIN {X 0,Y 131.094,Z 1047.191,A -85,B 0,C 180,E1 -25291.535,E2 -25291.535} C_VEL
LIN {X 0,Y 130.683,Z 1052.476,A -85,B 0,C 180,E1 -25294.626,E2 -25294.626} C_VEL
LIN {X 0,Y 130.058,Z 1058.586,A -85,B 0,C 180,E1 -25299.329,E2 -25299.329} C_VEL
LIN {X 0,Y 130.35,Z 1063.396,A -85,B 0,C 180,E1 -25303.957,E2 -25303.957} C_VEL
LIN {X 0,Y 131.818,Z 1067.334,A -85,B 0,C 180,E1 -25308.656,E2 -25308.656} C_VEL
LIN {X 0,Y 133.482,Z 1069.51,A -85,B 0,C 180,E1 -25311.626,E2 -25311.626} C_VEL
LIN {X 0,Y 138.145,Z 1072.473,A -85,B 0,C 180,E1 -25317.249,E2 -25317.249} C_VEL
LIN {X 0,Y 141.147,Z 1073.529,A -85,B 0,C 180,E1 -25319.862,E2 -25319.862} C_VEL
LIN {X 0,Y 148.526,Z 1074.388,A -85,B 0,C 180,E1 -25324.598,E2 -25324.598} C_VEL
LIN {X 0,Y 152.737,Z 1074.376,A -85,B 0,C 180,E1 -25326.739,E2 -25326.739} C_VEL
LIN {X 0,Y 162.156,Z 1073.033,A -85,B 0,C 180,E1 -25330.55,E2 -25330.55} C_VEL
LIN {X 0,Y 167.28,Z 1071.871,A -85,B 0,C 180,E1 -25332.238,E2 -25332.238} C_VEL
LIN {X 0,Y 175.411,Z 1069.286,A -85,B 0,C 180,E1 -25334.519,E2 -25334.519} C_VEL
LIN {X 0,Y 180.86,Z 1067.039,A -85,B 0,C 180,E1 -25335.83,E2 -25335.83} C_VEL
LIN {X 0,Y 180.415,Z 1067.116,A -85,B 0,C 180,E1 -25336.507,E2 -25336.507} C_VEL
LIN {X 0,Y 171.318,Z 1069.765,A -85,B 0,C 180,E1 -25338.978,E2 -25338.978} C_VEL
LIN {X 0,Y 166.071,Z 1070.808,A -85,B 0,C 180,E1 -25340.597,E2 -25340.597} C_VEL
LIN {X 0,Y 161.101,Z 1071.458,A -85,B 0,C 180,E1 -25342.358,E2 -25342.358} C_VEL
LIN {X 0,Y 151.972,Z 1071.356,A -85,B 0,C 180,E1 -25346.294,E2 -25346.294} C_VEL
LIN {X 0,Y 147.809,Z 1070.785,A -85,B 0,C 180,E1 -25348.466,E2 -25348.466} C_VEL
LIN {X 0,Y 140.567,Z 1068.274,A -85,B 0,C 180,E1 -25353.259,E2 -25353.259} C_VEL
LIN {X 0,Y 139.539,Z 1067.685,A -85,B 0,C 180,E1 -25354.116,E2 -25354.116} C_VEL
LIN {X 0,Y 136.631,Z 1066.091,A -85,B 0,C 180,E1 -25356.146,E2 -25356.146} C_VEL
LIN {X 0,Y 130.915,Z 1062.448,A -85,B 0,C 180,E1 -25359.279,E2 -25359.279} C_VEL
LIN {X 0,Y 125.916,Z 1058.084,A -85,B 0,C 180,E1 -25362.57,E2 -25362.57} C_VEL
LIN {X 0,Y 124.212,Z 1055.163,A -85,B 0,C 180,E1 -25364.792,E2 -25364.792} C_VEL
LIN {X 0,Y 122.784,Z 1048.08,A -85,B 0,C 180,E1 -25370.114,E2 -25370.114} C_VEL
LIN {X 0,Y 122.535,Z 1041.644,A -85,B 0,C 180,E1 -25374.241,E2 -25374.241} C_VEL
LIN {X 0,Y 122.69,Z 1033.641,A -85,B 0,C 180,E1 -25378.36,E2 -25378.36} C_VEL
LIN {X 0,Y 122.925,Z 1023.667,A -85,B 0,C 180,E1 -25382.459,E2 -25382.459} C_VEL
LIN {X 0,Y 123.401,Z 1013.488,A -85,B 0,C 180,E1 -25385.722,E2 -25385.722} C_VEL
LIN {X 0,Y 123.884,Z 1003.781,A -85,B 0,C 180,E1 -25388.155,E2 -25388.155} C_VEL
LIN {X 0,Y 124.494,Z 991.252,A -85,B 0,C 180,E1 -25390.574,E2 -25390.574} C_VEL
LIN {X 0,Y 124.71,Z 979.071,A -85,B 0,C 180,E1 -25392.202,E2 -25392.202} C_VEL
LIN {X 0,Y 125.481,Z 942.857,A -85,B 0,C 180,E1 -25396.564,E2 -25396.564} C_VEL
LIN {X 0,Y 125.57,Z 936.208,A -85,B 0,C 180,E1 -25397.333,E2 -25397.333} C_VEL
LIN {X 0,Y 123.417,Z 923.395,A -85,B 0,C 180,E1 -25398.618,E2 -25398.618} C_VEL
LIN {X 0,Y 122.844,Z 919.992,A -85,B 0,C 180,E1 -25399.006,E2 -25399.006} C_VEL
LIN {X 0,Y 121.964,Z 920.102,A -85,B 0,C 180,E1 -25407.453,E2 -25407.453} C_VEL
LIN {X 0,Y 121.899,Z 920.107,A -85,B 0,C 180,E1 -25411.26,E2 -25411.26} C_VEL
LIN {X 0,Y 121.882,Z 920.113,A -85,B 0,C 180,E1 -25416.17,E2 -25416.17} C_VEL
LIN {X 0,Y 121.864,Z 920.114,A -85,B 0,C 180,E1 -25421.435,E2 -25421.435} C_VEL
LIN {X 0,Y 121.865,Z 920.11,A -85,B 0,C 180,E1 -25428.568,E2 -25428.568} C_VEL
LIN {X 0,Y 121.909,Z 920.11,A -85,B 0,C 180,E1 -25434.796,E2 -25434.796} C_VEL
LIN {X 0,Y 121.929,Z 920.106,A -85,B 0,C 180,E1 -25439.841,E2 -25439.841} C_VEL
LIN {X 0,Y 121.955,Z 920.1,A -85,B 0,C 180,E1 -25446.21,E2 -25446.21} C_VEL
LIN {X 0,Y 121.993,Z 920.1,A -85,B 0,C 180,E1 -25449.779,E2 -25449.779} C_VEL
LIN {X 0,Y 122.191,Z 920.068,A -85,B 0,C 180,E1 -25456.7,E2 -25456.7} C_VEL
LIN {X 0,Y 122.4,Z 920.051,A -85,B 0,C 180,E1 -25460.082,E2 -25460.082} C_VEL
LIN {X 0,Y 122.551,Z 920.027,A -85,B 0,C 180,E1 -25466.713,E2 -25466.713} C_VEL
LIN {X 0,Y 123.018,Z 919.975,A -85,B 0,C 180,E1 -25470.001,E2 -25470.001} C_VEL
LIN {X 0,Y 122.407,Z 920.047,A -85,B 0,C 180,E1 -25476.594,E2 -25476.594} C_VEL
LIN {X 0,Y 122.399,Z 920.051,A -85,B 0,C 180,E1 -25479.92,E2 -25479.92} C_VEL
LIN {X 0,Y 122.19,Z 920.068,A -85,B 0,C 180,E1 -25483.302,E2 -25483.302} C_VEL
LIN {X 0,Y 121.99,Z 920.101,A -85,B 0,C 180,E1 -25490.223,E2 -25490.223} C_VEL
LIN {X 0,Y 121.915,Z 920.105,A -85,B 0,C 180,E1 -25493.8,E2 -25493.8} C_VEL
LIN {X 0,Y 121.919,Z 920.107,A -85,B 0,C 180,E1 -25500.151,E2 -25500.151} C_VEL
LIN {X 0,Y 121.884,Z 920.115,A -85,B 0,C 180,E1 -25506.168,E2 -25506.168} C_VEL
LIN {X 0,Y 121.867,Z 920.109,A -85,B 0,C 180,E1 -25511.433,E2 -25511.433} C_VEL
LIN {X 0,Y 121.866,Z 920.114,A -85,B 0,C 180,E1 -25518.566,E2 -25518.566} C_VEL
LIN {X 0,Y 121.911,Z 920.112,A -85,B 0,C 180,E1 -25524.794,E2 -25524.794} C_VEL
LIN {X 0,Y 121.919,Z 920.102,A -85,B 0,C 180,E1 -25529.847,E2 -25529.847} C_VEL
LIN {X 0,Y 121.982,Z 920.099,A -85,B 0,C 180,E1 -25537.199,E2 -25537.199} C_VEL
LIN {X 0,Y 122.062,Z 920.094,A -85,B 0,C 180,E1 -25543.267,E2 -25543.267} C_VEL
LIN {X 0,Y 122.289,Z 920.056,A -85,B 0,C 180,E1 -25547.69,E2 -25547.69} C_VEL
LIN {X 0,Y 122.398,Z 920.047,A -85,B 0,C 180,E1 -25550.079,E2 -25550.079} C_VEL
LIN {X 0,Y 122.549,Z 920.026,A -85,B 0,C 180,E1 -25556.711,E2 -25556.711} C_VEL
LIN {X 0,Y 123.016,Z 919.971,A -85,B 0,C 180,E1 -25559.998,E2 -25559.998} C_VEL
LIN {X 0,Y 122.4,Z 920.043,A -85,B 0,C 180,E1 -25566.593,E2 -25566.593} C_VEL
LIN {X 0,Y 122.391,Z 920.05,A -85,B 0,C 180,E1 -25569.918,E2 -25569.918} C_VEL
LIN {X 0,Y 122.188,Z 920.075,A -85,B 0,C 180,E1 -25573.3,E2 -25573.3} C_VEL
LIN {X 0,Y 121.987,Z 920.101,A -85,B 0,C 180,E1 -25580.222,E2 -25580.222} C_VEL
LIN {X 0,Y 121.911,Z 920.107,A -85,B 0,C 180,E1 -25583.798,E2 -25583.798} C_VEL
LIN {X 0,Y 121.915,Z 920.11,A -85,B 0,C 180,E1 -25590.15,E2 -25590.15} C_VEL
LIN {X 0,Y 121.88,Z 920.112,A -85,B 0,C 180,E1 -25596.167,E2 -25596.167} C_VEL
LIN {X 0,Y 121.862,Z 920.116,A -85,B 0,C 180,E1 -25601.432,E2 -25601.432} C_VEL
LIN {X 0,Y 121.862,Z 920.118,A -85,B 0,C 180,E1 -25608.565,E2 -25608.565} C_VEL
LIN {X 0,Y 121.934,Z 920.105,A -85,B 0,C 180,E1 -25614.803,E2 -25614.803} C_VEL
LIN {X 0,Y 122.466,Z 920.035,A -85,B 0,C 180,E1 -25622.67,E2 -25622.67} C_VEL
LIN {X 0,Y 122.773,Z 920.006,A -85,B 0,C 180,E1 -25626.377,E2 -25626.377} C_VEL
LIN {X 0,Y 122.519,Z 920.037,A -85,B 0,C 180,E1 -25629.758,E2 -25629.758} C_VEL
LIN {X 0,Y 122.97,Z 938.461,A -85,B 0,C 180,E1 -25631.894,E2 -25631.894} C_VEL
LIN {X 0,Y 125.376,Z 964.063,A -85,B 0,C 180,E1 -25634.635,E2 -25634.635} C_VEL
LIN {X 0,Y 125.589,Z 971.718,A -85,B 0,C 180,E1 -25635.518,E2 -25635.518} C_VEL
LIN {X 0,Y 125.335,Z 998.515,A -85,B 0,C 180,E1 -25638.886,E2 -25638.886} C_VEL
LIN {X 0,Y 125.063,Z 1010.999,A -85,B 0,C 180,E1 -25641.109,E2 -25641.109} C_VEL
LIN {X 0,Y 124.866,Z 1021.077,A -85,B 0,C 180,E1 -25643.536,E2 -25643.536} C_VEL
LIN {X 0,Y 124.689,Z 1030.4,A -85,B 0,C 180,E1 -25646.364,E2 -25646.364} C_VEL
LIN {X 0,Y 124.693,Z 1037.959,A -85,B 0,C 180,E1 -25649.192,E2 -25649.192} C_VEL
LIN {X 0,Y 124.678,Z 1044.864,A -85,B 0,C 180,E1 -25652.422,E2 -25652.422} C_VEL
LIN {X 0,Y 124.255,Z 1050.238,A -85,B 0,C 180,E1 -25655.68,E2 -25655.68} C_VEL
LIN {X 0,Y 123.691,Z 1057.525,A -85,B 0,C 180,E1 -25661.47,E2 -25661.47} C_VEL
LIN {X 0,Y 124.321,Z 1062.37,A -85,B 0,C 180,E1 -25666.418,E2 -25666.418} C_VEL
LIN {X 0,Y 126.277,Z 1066.313,A -85,B 0,C 180,E1 -25671.208,E2 -25671.208} C_VEL
LIN {X 0,Y 129.441,Z 1069.4,A -85,B 0,C 180,E1 -25675.744,E2 -25675.744} C_VEL
LIN {X 0,Y 132.004,Z 1071.017,A -85,B 0,C 180,E1 -25678.631,E2 -25678.631} C_VEL
LIN {X 0,Y 138.736,Z 1073.13,A -85,B 0,C 180,E1 -25683.864,E2 -25683.864} C_VEL
LIN {X 0,Y 142.765,Z 1073.713,A -85,B 0,C 180,E1 -25686.209,E2 -25686.209} C_VEL
LIN {X 0,Y 151.798,Z 1073.807,A -85,B 0,C 180,E1 -25690.404,E2 -25690.404} C_VEL
LIN {X 0,Y 162.084,Z 1072.377,A -85,B 0,C 180,E1 -25693.928,E2 -25693.928} C_VEL
LIN {X 0,Y 168.839,Z 1070.8,A -85,B 0,C 180,E1 -25695.797,E2 -25695.797} C_VEL
LIN {X 0,Y 169.143,Z 1070.617,A -85,B 0,C 180,E1 -25696.538,E2 -25696.538} C_VEL
LIN {X 0,Y 160.681,Z 1071.853,A -85,B 0,C 180,E1 -25699,E2 -25699} C_VEL
LIN {X 0,Y 150.68,Z 1071.952,A -85,B 0,C 180,E1 -25702.676,E2 -25702.676} C_VEL
LIN {X 0,Y 146.121,Z 1071.412,A -85,B 0,C 180,E1 -25704.75,E2 -25704.75} C_VEL
LIN {X 0,Y 137.909,Z 1069.139,A -85,B 0,C 180,E1 -25709.364,E2 -25709.364} C_VEL
LIN {X 0,Y 132.734,Z 1066.416,A -85,B 0,C 180,E1 -25713.254,E2 -25713.254} C_VEL
LIN {X 0,Y 128.604,Z 1062.784,A -85,B 0,C 180,E1 -25717.511,E2 -25717.511} C_VEL
LIN {X 0,Y 125.565,Z 1058.204,A -85,B 0,C 180,E1 -25722.083,E2 -25722.083} C_VEL
LIN {X 0,Y 124.212,Z 1055.163,A -85,B 0,C 180,E1 -25724.792,E2 -25724.792} C_VEL
LIN {X 0,Y 122.831,Z 1052.047,A -85,B 0,C 180,E1 -25726.991,E2 -25726.991} C_VEL
LIN {X 0,Y 119.53,Z 1045.972,A -85,B 0,C 180,E1 -25730.321,E2 -25730.321} C_VEL
LIN {X 0,Y 116.691,Z 1039.137,A -85,B 0,C 180,E1 -25733.613,E2 -25733.613} C_VEL
LIN {X 0,Y 116.121,Z 1034.894,A -85,B 0,C 180,E1 -25735.709,E2 -25735.709} C_VEL
LIN {X 0,Y 116.218,Z 1028.64,A -85,B 0,C 180,E1 -25738.702,E2 -25738.702} C_VEL
LIN {X 0,Y 116.489,Z 1019.766,A -85,B 0,C 180,E1 -25742.163,E2 -25742.163} C_VEL
LIN {X 0,Y 116.932,Z 1008.767,A -85,B 0,C 180,E1 -25745.607,E2 -25745.607} C_VEL
LIN {X 0,Y 117.465,Z 996.87,A -85,B 0,C 180,E1 -25748.387,E2 -25748.387} C_VEL
LIN {X 0,Y 117.866,Z 986.64,A -85,B 0,C 180,E1 -25750.198,E2 -25750.198} C_VEL
LIN {X 0,Y 118.482,Z 946.817,A -85,B 0,C 180,E1 -25755.373,E2 -25755.373} C_VEL
LIN {X 0,Y 118.559,Z 936.139,A -85,B 0,C 180,E1 -25756.688,E2 -25756.688} C_VEL
LIN {X 0,Y 116.339,Z 923.169,A -85,B 0,C 180,E1 -25758.054,E2 -25758.054} C_VEL
LIN {X 0,Y 115.918,Z 920.858,A -85,B 0,C 180,E1 -25758.402,E2 -25758.402} C_VEL
LIN {X 0,Y 114.968,Z 920.977,A -85,B 0,C 180,E1 -25765.337,E2 -25765.337} C_VEL
LIN {X 0,Y 114.856,Z 920.983,A -85,B 0,C 180,E1 -25771.058,E2 -25771.058} C_VEL
LIN {X 0,Y 114.776,Z 920.995,A -85,B 0,C 180,E1 -25777.76,E2 -25777.76} C_VEL
LIN {X 0,Y 114.779,Z 920.999,A -85,B 0,C 180,E1 -25782.713,E2 -25782.713} C_VEL
LIN {X 0,Y 114.788,Z 920.992,A -85,B 0,C 180,E1 -25787.664,E2 -25787.664} C_VEL
LIN {X 0,Y 114.785,Z 920.999,A -85,B 0,C 180,E1 -25792.749,E2 -25792.749} C_VEL
LIN {X 0,Y 114.857,Z 920.984,A -85,B 0,C 180,E1 -25798.946,E2 -25798.946} C_VEL
LIN {X 0,Y 114.918,Z 920.975,A -85,B 0,C 180,E1 -25806.547,E2 -25806.547} C_VEL
LIN {X 0,Y 114.971,Z 920.975,A -85,B 0,C 180,E1 -25812.204,E2 -25812.204} C_VEL
LIN {X 0,Y 115.313,Z 920.933,A -85,B 0,C 180,E1 -25819.465,E2 -25819.465} C_VEL
LIN {X 0,Y 115.479,Z 920.907,A -85,B 0,C 180,E1 -25826.511,E2 -25826.511} C_VEL
LIN {X 0,Y 115.946,Z 920.856,A -85,B 0,C 180,E1 -25830.001,E2 -25830.001} C_VEL
LIN {X 0,Y 115.35,Z 920.927,A -85,B 0,C 180,E1 -25837,E2 -25837} C_VEL
LIN {X 0,Y 115.208,Z 920.94,A -85,B 0,C 180,E1 -25842.558,E2 -25842.558} C_VEL
LIN {X 0,Y 114.967,Z 920.976,A -85,B 0,C 180,E1 -25847.798,E2 -25847.798} C_VEL
LIN {X 0,Y 114.897,Z 920.978,A -85,B 0,C 180,E1 -25853.429,E2 -25853.429} C_VEL
LIN {X 0,Y 114.85,Z 920.985,A -85,B 0,C 180,E1 -25861.049,E2 -25861.049} C_VEL
LIN {X 0,Y 114.778,Z 921,A -85,B 0,C 180,E1 -25867.758,E2 -25867.758} C_VEL
LIN {X 0,Y 114.782,Z 920.995,A -85,B 0,C 180,E1 -25872.711,E2 -25872.711} C_VEL
LIN {X 0,Y 114.789,Z 920.998,A -85,B 0,C 180,E1 -25877.662,E2 -25877.662} C_VEL
LIN {X 0,Y 114.787,Z 920.996,A -85,B 0,C 180,E1 -25882.746,E2 -25882.746} C_VEL
LIN {X 0,Y 114.85,Z 920.984,A -85,B 0,C 180,E1 -25888.95,E2 -25888.95} C_VEL
LIN {X 0,Y 114.902,Z 920.984,A -85,B 0,C 180,E1 -25896.563,E2 -25896.563} C_VEL
LIN {X 0,Y 114.967,Z 920.975,A -85,B 0,C 180,E1 -25902.201,E2 -25902.201} C_VEL
LIN {X 0,Y 115.311,Z 920.926,A -85,B 0,C 180,E1 -25909.463,E2 -25909.463} C_VEL
LIN {X 0,Y 115.476,Z 920.907,A -85,B 0,C 180,E1 -25916.509,E2 -25916.509} C_VEL
LIN {X 0,Y 115.944,Z 920.852,A -85,B 0,C 180,E1 -25919.998,E2 -25919.998} C_VEL
LIN {X 0,Y 115.343,Z 920.921,A -85,B 0,C 180,E1 -25926.998,E2 -25926.998} C_VEL
LIN {X 0,Y 115.205,Z 920.947,A -85,B 0,C 180,E1 -25932.556,E2 -25932.556} C_VEL
LIN {X 0,Y 114.965,Z 920.972,A -85,B 0,C 180,E1 -25937.796,E2 -25937.796} C_VEL
LIN {X 0,Y 114.893,Z 920.981,A -85,B 0,C 180,E1 -25943.427,E2 -25943.427} C_VEL
LIN {X 0,Y 114.847,Z 920.992,A -85,B 0,C 180,E1 -25951.048,E2 -25951.048} C_VEL
LIN {X 0,Y 114.774,Z 921,A -85,B 0,C 180,E1 -25957.757,E2 -25957.757} C_VEL
LIN {X 0,Y 114.777,Z 920.994,A -85,B 0,C 180,E1 -25962.71,E2 -25962.71} C_VEL
LIN {X 0,Y 114.785,Z 920.999,A -85,B 0,C 180,E1 -25967.661,E2 -25967.661} C_VEL
LIN {X 0,Y 114.794,Z 920.99,A -85,B 0,C 180,E1 -25972.737,E2 -25972.737} C_VEL
LIN {X 0,Y 115.199,Z 920.942,A -85,B 0,C 180,E1 -25980.786,E2 -25980.786} C_VEL
LIN {X 0,Y 115.639,Z 920.895,A -85,B 0,C 180,E1 -25985.728,E2 -25985.728} C_VEL
LIN {X 0,Y 115.543,Z 920.907,A -85,B 0,C 180,E1 -25990.455,E2 -25990.455} C_VEL
LIN {X 0,Y 116.124,Z 940.31,A -85,B 0,C 180,E1 -25992.824,E2 -25992.824} C_VEL
LIN {X 0,Y 118.775,Z 967.655,A -85,B 0,C 180,E1 -25995.928,E2 -25995.928} C_VEL
LIN {X 0,Y 118.652,Z 997.436,A -85,B 0,C 180,E1 -25999.871,E2 -25999.871} C_VEL
LIN {X 0,Y 118.441,Z 1008.644,A -85,B 0,C 180,E1 -26001.898,E2 -26001.898} C_VEL
LIN {X 0,Y 118.317,Z 1019.03,A -85,B 0,C 180,E1 -26004.46,E2 -26004.46} C_VEL
LIN {X 0,Y 118.264,Z 1028.421,A -85,B 0,C 180,E1 -26007.445,E2 -26007.445} C_VEL
